LIN {X 0,Y 354.479,Z 638.418,A -85,B 0,C 180,E1 -13745.915,E2 -13745.915} C_VEL
LIN {X 0,Y 358.461,Z 680.686,A -85,B 0,C 180,E1 -13747.67,E2 -13747.67} C_VEL
LIN {X 0,Y 356.651,Z 726.677,A -85,B 0,C 180,E1 -13748.951,E2 -13748.951} C_VEL
LIN {X 0,Y 355.646,Z 740.597,A -85,B 0,C 180,E1 -13749.542,E2 -13749.542} C_VEL
LIN {X 0,Y 354.363,Z 753.48,A -85,B 0,C 180,E1 -13750.297,E2 -13750.297} C_VEL
LIN {X 0,Y 352.622,Z 767.795,A -85,B 0,C 180,E1 -13751.405,E2 -13751.405} C_VEL
LIN {X 0,Y 351.171,Z 779.191,A -85,B 0,C 180,E1 -13752.531,E2 -13752.531} C_VEL
LIN {X 0,Y 349.769,Z 790.795,A -85,B 0,C 180,E1 -13753.962,E2 -13753.962} C_VEL
LIN {X 0,Y 348.561,Z 801.445,A -85,B 0,C 180,E1 -13755.583,E2 -13755.583} C_VEL
LIN {X 0,Y 347.802,Z 809.876,A -85,B 0,C 180,E1 -13757.158,E2 -13757.158} C_VEL
LIN {X 0,Y 347.231,Z 817.648,A -85,B 0,C 180,E1 -13758.915,E2 -13758.915} C_VEL
LIN {X 0,Y 347.018,Z 823.966,A -85,B 0,C 180,E1 -13760.677,E2 -13760.677} C_VEL
LIN {X 0,Y 347.018,Z 831.536,A -85,B 0,C 180,E1 -13763.321,E2 -13763.321} C_VEL
LIN {X 0,Y 347.321,Z 835.911,A -85,B 0,C 180,E1 -13765.358,E2 -13765.358} C_VEL
LIN {X 0,Y 347.318,Z 837.708,A -85,B 0,C 180,E1 -13766.52,E2 -13766.52} C_VEL
LIN {X 0,Y 347.353,Z 838.988,A -85,B 0,C 180,E1 -13767.682,E2 -13767.682} C_VEL
LIN {X 0,Y 347.487,Z 839.813,A -85,B 0,C 180,E1 -13768.842,E2 -13768.842} C_VEL
LIN {X 0,Y 347.688,Z 840.196,A -85,B 0,C 180,E1 -13770.001,E2 -13770.001} C_VEL
LIN {X 0,Y 347.364,Z 840.046,A -85,B 0,C 180,E1 -13771.16,E2 -13771.16} C_VEL
LIN {X 0,Y 347.277,Z 839.445,A -85,B 0,C 180,E1 -13772.32,E2 -13772.32} C_VEL
LIN {X 0,Y 347.224,Z 838.385,A -85,B 0,C 180,E1 -13773.482,E2 -13773.482} C_VEL
LIN {X 0,Y 347.158,Z 836.872,A -85,B 0,C 180,E1 -13774.645,E2 -13774.645} C_VEL
LIN {X 0,Y 346.924,Z 833.32,A -85,B 0,C 180,E1 -13776.582,E2 -13776.582} C_VEL
LIN {X 0,Y 346.84,Z 827.807,A -85,B 0,C 180,E1 -13778.742,E2 -13778.742} C_VEL
LIN {X 0,Y 347.027,Z 820.861,A -85,B 0,C 180,E1 -13780.798,E2 -13780.798} C_VEL
LIN {X 0,Y 347.607,Z 813.484,A -85,B 0,C 180,E1 -13782.554,E2 -13782.554} C_VEL
LIN {X 0,Y 348.199,Z 805.239,A -85,B 0,C 180,E1 -13784.184,E2 -13784.184} C_VEL
LIN {X 0,Y 349.492,Z 795.668,A -85,B 0,C 180,E1 -13785.753,E2 -13785.753} C_VEL
LIN {X 0,Y 350.936,Z 785.164,A -85,B 0,C 180,E1 -13787.182,E2 -13787.182} C_VEL
LIN {X 0,Y 352.74,Z 772.484,A -85,B 0,C 180,E1 -13788.59,E2 -13788.59} C_VEL
LIN {X 0,Y 354.368,Z 760.134,A -85,B 0,C 180,E1 -13789.704,E2 -13789.704} C_VEL
LIN {X 0,Y 356.324,Z 745.84,A -85,B 0,C 180,E1 -13790.72,E2 -13790.72} C_VEL
LIN {X 0,Y 358.072,Z 729.548,A -85,B 0,C 180,E1 -13791.594,E2 -13791.594} C_VEL
LIN {X 0,Y 359.248,Z 714.539,A -85,B 0,C 180,E1 -13792.171,E2 -13792.171} C_VEL
LIN {X 0,Y 360.847,Z 679.966,A -85,B 0,C 180,E1 -13793.198,E2 -13793.198} C_VEL
LIN {X 0,Y 359.795,Z 647.693,A -85,B 0,C 180,E1 -13794.475,E2 -13794.475} C_VEL
LIN {X 0,Y 358.265,Z 629.878,A -85,B 0,C 180,E1 -13795.336,E2 -13795.336} C_VEL
LIN {X 0,Y 355.685,Z 611.993,A -85,B 0,C 180,E1 -13796.387,E2 -13796.387} C_VEL
LIN {X 0,Y 353.303,Z 598.764,A -85,B 0,C 180,E1 -13797.284,E2 -13797.284} C_VEL
LIN {X 0,Y 350.384,Z 585.333,A -85,B 0,C 180,E1 -13798.328,E2 -13798.328} C_VEL
LIN {X 0,Y 349.237,Z 579.78,A -85,B 0,C 180,E1 -13798.781,E2 -13798.781} C_VEL
LIN {X 0,Y 349.199,Z 578.981,A -85,B 0,C 180,E1 -13798.884,E2 -13798.884} C_VEL
LIN {X 0,Y 349.844,Z 568.142,A -85,B 0,C 180,E1 -13801.488,E2 -13801.488} C_VEL
LIN {X 0,Y 347.976,Z 557.739,A -85,B 0,C 180,E1 -13804.286,E2 -13804.286} C_VEL
LIN {X 0,Y 347.852,Z 557.158,A -85,B 0,C 180,E1 -13804.452,E2 -13804.452} C_VEL
LIN {X 0,Y 347.778,Z 557.162,A -85,B 0,C 180,E1 -13807.989,E2 -13807.989} C_VEL
LIN {X 0,Y 347.755,Z 557.164,A -85,B 0,C 180,E1 -13811.83,E2 -13811.83} C_VEL
LIN {X 0,Y 347.71,Z 557.174,A -85,B 0,C 180,E1 -13815.027,E2 -13815.027} C_VEL
LIN {X 0,Y 347.755,Z 557.165,A -85,B 0,C 180,E1 -13818.397,E2 -13818.397} C_VEL
LIN {X 0,Y 347.778,Z 557.163,A -85,B 0,C 180,E1 -13822.011,E2 -13822.011} C_VEL
LIN {X 0,Y 347.749,Z 557.169,A -85,B 0,C 180,E1 -13825.536,E2 -13825.536} C_VEL
LIN {X 0,Y 347.749,Z 557.167,A -85,B 0,C 180,E1 -13828.3,E2 -13828.3} C_VEL
LIN {X 0,Y 347.825,Z 557.277,A -85,B 0,C 180,E1 -13831.453,E2 -13831.453} C_VEL
LIN {X 0,Y 348.808,Z 559.969,A -85,B 0,C 180,E1 -13831.741,E2 -13831.741} C_VEL
LIN {X 0,Y 351.052,Z 562.747,A -85,B 0,C 180,E1 -13832.234,E2 -13832.234} C_VEL
LIN {X 0,Y 353.196,Z 565.986,A -85,B 0,C 180,E1 -13832.701,E2 -13832.701} C_VEL
LIN {X 0,Y 358.206,Z 574.137,A -85,B 0,C 180,E1 -13833.732,E2 -13833.732} C_VEL
LIN {X 0,Y 363.446,Z 583.854,A -85,B 0,C 180,E1 -13834.746,E2 -13834.746} C_VEL
LIN {X 0,Y 365.343,Z 588.205,A -85,B 0,C 180,E1 -13835.107,E2 -13835.107} C_VEL
LIN {X 0,Y 364.896,Z 614.714,A -85,B 0,C 180,E1 -13835.837,E2 -13835.837} C_VEL
LIN {X 0,Y 364.662,Z 629.49,A -85,B 0,C 180,E1 -13836.415,E2 -13836.415} C_VEL
LIN {X 0,Y 364.052,Z 644.188,A -85,B 0,C 180,E1 -13837.22,E2 -13837.22} C_VEL
LIN {X 0,Y 363.117,Z 657.203,A -85,B 0,C 180,E1 -13838.155,E2 -13838.155} C_VEL
LIN {X 0,Y 361.975,Z 669.32,A -85,B 0,C 180,E1 -13839.249,E2 -13839.249} C_VEL
LIN {X 0,Y 360.436,Z 681.905,A -85,B 0,C 180,E1 -13840.641,E2 -13840.641} C_VEL
LIN {X 0,Y 358.957,Z 692.336,A -85,B 0,C 180,E1 -13842.039,E2 -13842.039} C_VEL
LIN {X 0,Y 357.274,Z 702.674,A -85,B 0,C 180,E1 -13843.721,E2 -13843.721} C_VEL
LIN {X 0,Y 355.557,Z 712.086,A -85,B 0,C 180,E1 -13845.593,E2 -13845.593} C_VEL
LIN {X 0,Y 353.869,Z 720.615,A -85,B 0,C 180,E1 -13847.672,E2 -13847.672} C_VEL
LIN {X 0,Y 352.478,Z 727.173,A -85,B 0,C 180,E1 -13849.662,E2 -13849.662} C_VEL
LIN {X 0,Y 351.014,Z 733.098,A -85,B 0,C 180,E1 -13851.943,E2 -13851.943} C_VEL
LIN {X 0,Y 350.103,Z 737.454,A -85,B 0,C 180,E1 -13854.239,E2 -13854.239} C_VEL
LIN {X 0,Y 349.236,Z 740.513,A -85,B 0,C 180,E1 -13856.538,E2 -13856.538} C_VEL
LIN {X 0,Y 348.701,Z 742.261,A -85,B 0,C 180,E1 -13858.845,E2 -13858.845} C_VEL
LIN {X 0,Y 348.344,Z 742.765,A -85,B 0,C 180,E1 -13861.156,E2 -13861.156} C_VEL
LIN {X 0,Y 348.06,Z 742.044,A -85,B 0,C 180,E1 -13863.472,E2 -13863.472} C_VEL
LIN {X 0,Y 348.044,Z 740.07,A -85,B 0,C 180,E1 -13865.794,E2 -13865.794} C_VEL
LIN {X 0,Y 348.199,Z 738.597,A -85,B 0,C 180,E1 -13866.955,E2 -13866.955} C_VEL
LIN {X 0,Y 348.351,Z 734.679,A -85,B 0,C 180,E1 -13869.288,E2 -13869.288} C_VEL
LIN {X 0,Y 348.678,Z 729.336,A -85,B 0,C 180,E1 -13871.628,E2 -13871.628} C_VEL
LIN {X 0,Y 349.239,Z 722.409,A -85,B 0,C 180,E1 -13873.974,E2 -13873.974} C_VEL
LIN {X 0,Y 349.954,Z 714.96,A -85,B 0,C 180,E1 -13875.999,E2 -13875.999} C_VEL
LIN {X 0,Y 350.859,Z 705.636,A -85,B 0,C 180,E1 -13878.087,E2 -13878.087} C_VEL
LIN {X 0,Y 351.878,Z 695.29,A -85,B 0,C 180,E1 -13880,E2 -13880} C_VEL
LIN {X 0,Y 352.954,Z 683.746,A -85,B 0,C 180,E1 -13881.768,E2 -13881.768} C_VEL
LIN {X 0,Y 354.106,Z 670.886,A -85,B 0,C 180,E1 -13883.387,E2 -13883.387} C_VEL
LIN {X 0,Y 355.051,Z 658.101,A -85,B 0,C 180,E1 -13884.718,E2 -13884.718} C_VEL
LIN {X 0,Y 356.033,Z 644.114,A -85,B 0,C 180,E1 -13885.896,E2 -13885.896} C_VEL
LIN {X 0,Y 356.796,Z 629.668,A -85,B 0,C 180,E1 -13886.859,E2 -13886.859} C_VEL
LIN {X 0,Y 357.368,Z 614.609,A -85,B 0,C 180,E1 -13887.621,E2 -13887.621} C_VEL
LIN {X 0,Y 357.586,Z 599.377,A -85,B 0,C 180,E1 -13888.166,E2 -13888.166} C_VEL
LIN {X 0,Y 357.616,Z 583.757,A -85,B 0,C 180,E1 -13888.584,E2 -13888.584} C_VEL
LIN {X 0,Y 347.819,Z 557.232,A -85,B 0,C 180,E1 -13889.822,E2 -13889.822} C_VEL
LIN {X 0,Y 347.749,Z 557.17,A -85,B 0,C 180,E1 -13894.043,E2 -13894.043} C_VEL
LIN {X 0,Y 347.762,Z 557.162,A -85,B 0,C 180,E1 -13897.32,E2 -13897.32} C_VEL
LIN {X 0,Y 347.733,Z 557.172,A -85,B 0,C 180,E1 -13900.296,E2 -13900.296} C_VEL
LIN {X 0,Y 347.723,Z 557.167,A -85,B 0,C 180,E1 -13903.407,E2 -13903.407} C_VEL
LIN {X 0,Y 347.725,Z 557.17,A -85,B 0,C 180,E1 -13906.685,E2 -13906.685} C_VEL
LIN {X 0,Y 347.747,Z 557.168,A -85,B 0,C 180,E1 -13910.172,E2 -13910.172} C_VEL
LIN {X 0,Y 347.766,Z 557.166,A -85,B 0,C 180,E1 -13912.679,E2 -13912.679} C_VEL
LIN {X 0,Y 347.748,Z 557.165,A -85,B 0,C 180,E1 -13915.955,E2 -13915.955} C_VEL
LIN {X 0,Y 347.748,Z 557.164,A -85,B 0,C 180,E1 -13919.651,E2 -13919.651} C_VEL
LIN {X 0,Y 347.83,Z 557.154,A -85,B 0,C 180,E1 -13923.607,E2 -13923.607} C_VEL
LIN {X 0,Y 347.788,Z 557.161,A -85,B 0,C 180,E1 -13926.161,E2 -13926.161} C_VEL
LIN {X 0,Y 347.811,Z 557.156,A -85,B 0,C 180,E1 -13929.909,E2 -13929.909} C_VEL
LIN {X 0,Y 347.865,Z 557.152,A -85,B 0,C 180,E1 -13932.359,E2 -13932.359} C_VEL
LIN {X 0,Y 347.896,Z 557.146,A -85,B 0,C 180,E1 -13935.97,E2 -13935.97} C_VEL
LIN {X 0,Y 347.927,Z 557.143,A -85,B 0,C 180,E1 -13939.525,E2 -13939.525} C_VEL
LIN {X 0,Y 348.072,Z 557.124,A -85,B 0,C 180,E1 -13941.874,E2 -13941.874} C_VEL
LIN {X 0,Y 348.066,Z 557.125,A -85,B 0,C 180,E1 -13944.205,E2 -13944.205} C_VEL
LIN {X 0,Y 348.206,Z 557.108,A -85,B 0,C 180,E1 -13947.686,E2 -13947.686} C_VEL
LIN {X 0,Y 348.344,Z 557.09,A -85,B 0,C 180,E1 -13949.999,E2 -13949.999} C_VEL
LIN {X 0,Y 348.206,Z 557.107,A -85,B 0,C 180,E1 -13952.313,E2 -13952.313} C_VEL
LIN {X 0,Y 348.101,Z 557.123,A -85,B 0,C 180,E1 -13956.957,E2 -13956.957} C_VEL
LIN {X 0,Y 347.965,Z 557.144,A -85,B 0,C 180,E1 -13959.298,E2 -13959.298} C_VEL
LIN {X 0,Y 347.891,Z 557.148,A -85,B 0,C 180,E1 -13962.839,E2 -13962.839} C_VEL
LIN {X 0,Y 347.836,Z 557.153,A -85,B 0,C 180,E1 -13966.431,E2 -13966.431} C_VEL
LIN {X 0,Y 347.847,Z 557.153,A -85,B 0,C 180,E1 -13968.86,E2 -13968.86} C_VEL
LIN {X 0,Y 347.771,Z 557.161,A -85,B 0,C 180,E1 -13972.579,E2 -13972.579} C_VEL
LIN {X 0,Y 347.808,Z 557.158,A -85,B 0,C 180,E1 -13975.108,E2 -13975.108} C_VEL
LIN {X 0,Y 347.808,Z 557.163,A -85,B 0,C 180,E1 -13977.693,E2 -13977.693} C_VEL
LIN {X 0,Y 347.767,Z 557.163,A -85,B 0,C 180,E1 -13980.345,E2 -13980.345} C_VEL
LIN {X 0,Y 347.743,Z 557.168,A -85,B 0,C 180,E1 -13984.043,E2 -13984.043} C_VEL
LIN {X 0,Y 347.761,Z 557.164,A -85,B 0,C 180,E1 -13987.32,E2 -13987.32} C_VEL
LIN {X 0,Y 347.75,Z 557.166,A -85,B 0,C 180,E1 -13990.294,E2 -13990.294} C_VEL
LIN {X 0,Y 347.764,Z 557.164,A -85,B 0,C 180,E1 -13993.401,E2 -13993.401} C_VEL
LIN {X 0,Y 347.809,Z 557.157,A -85,B 0,C 180,E1 -13996.67,E2 -13996.67} C_VEL
LIN {X 0,Y 347.78,Z 557.165,A -85,B 0,C 180,E1 -14000.123,E2 -14000.123} C_VEL
LIN {X 0,Y 347.68,Z 557.818,A -85,B 0,C 180,E1 -14000.73,E2 -14000.73} C_VEL
LIN {X 0,Y 347.391,Z 559.998,A -85,B 0,C 180,E1 -14001.422,E2 -14001.422} C_VEL
LIN {X 0,Y 347.087,Z 563.175,A -85,B 0,C 180,E1 -14002.021,E2 -14002.021} C_VEL
LIN {X 0,Y 346.917,Z 567.944,A -85,B 0,C 180,E1 -14002.622,E2 -14002.622} C_VEL
LIN {X 0,Y 347.234,Z 573.312,A -85,B 0,C 180,E1 -14003.094,E2 -14003.094} C_VEL
LIN {X 0,Y 348.465,Z 578.915,A -85,B 0,C 180,E1 -14003.416,E2 -14003.416} C_VEL
LIN {X 0,Y 349.772,Z 582.501,A -85,B 0,C 180,E1 -14003.573,E2 -14003.573} C_VEL
LIN {X 0,Y 349.053,Z 620.126,A -85,B 0,C 180,E1 -14004.541,E2 -14004.541} C_VEL
LIN {X 0,Y 348.82,Z 634.327,A -85,B 0,C 180,E1 -14005.132,E2 -14005.132} C_VEL
LIN {X 0,Y 348.195,Z 648.532,A -85,B 0,C 180,E1 -14005.963,E2 -14005.963} C_VEL
LIN {X 0,Y 347.478,Z 660.802,A -85,B 0,C 180,E1 -14006.901,E2 -14006.901} C_VEL
LIN {X 0,Y 346.554,Z 674.042,A -85,B 0,C 180,E1 -14008.179,E2 -14008.179} C_VEL
LIN {X 0,Y 345.474,Z 685.971,A -85,B 0,C 180,E1 -14009.601,E2 -14009.601} C_VEL
LIN {X 0,Y 344.643,Z 696.152,A -85,B 0,C 180,E1 -14011.089,E2 -14011.089} C_VEL
LIN {X 0,Y 343.596,Z 706.515,A -85,B 0,C 180,E1 -14012.929,E2 -14012.929} C_VEL
LIN {X 0,Y 342.781,Z 715.232,A -85,B 0,C 180,E1 -14014.822,E2 -14014.822} C_VEL
LIN {X 0,Y 342.118,Z 722.337,A -85,B 0,C 180,E1 -14016.707,E2 -14016.707} C_VEL
LIN {X 0,Y 341.513,Z 728.954,A -85,B 0,C 180,E1 -14018.892,E2 -14018.892} C_VEL
LIN {X 0,Y 341.151,Z 733.355,A -85,B 0,C 180,E1 -14020.755,E2 -14020.755} C_VEL
LIN {X 0,Y 340.967,Z 735.707,A -85,B 0,C 180,E1 -14021.991,E2 -14021.991} C_VEL
LIN {X 0,Y 340.772,Z 739.15,A -85,B 0,C 180,E1 -14024.449,E2 -14024.449} C_VEL
LIN {X 0,Y 340.83,Z 741.068,A -85,B 0,C 180,E1 -14026.89,E2 -14026.89} C_VEL
LIN {X 0,Y 340.94,Z 741.459,A -85,B 0,C 180,E1 -14028.105,E2 -14028.105} C_VEL
LIN {X 0,Y 341.317,Z 741.079,A -85,B 0,C 180,E1 -14030.519,E2 -14030.519} C_VEL
LIN {X 0,Y 341.831,Z 739.281,A -85,B 0,C 180,E1 -14032.915,E2 -14032.915} C_VEL
LIN {X 0,Y 342.719,Z 735.987,A -85,B 0,C 180,E1 -14035.295,E2 -14035.295} C_VEL
LIN {X 0,Y 343.442,Z 732.461,A -85,B 0,C 180,E1 -14037.068,E2 -14037.068} C_VEL
LIN {X 0,Y 344.428,Z 727.73,A -85,B 0,C 180,E1 -14038.915,E2 -14038.915} C_VEL
LIN {X 0,Y 345.636,Z 721.395,A -85,B 0,C 180,E1 -14040.874,E2 -14040.874} C_VEL
LIN {X 0,Y 346.918,Z 714.409,A -85,B 0,C 180,E1 -14042.613,E2 -14042.613} C_VEL
LIN {X 0,Y 348.453,Z 705.922,A -85,B 0,C 180,E1 -14044.338,E2 -14044.338} C_VEL
LIN {X 0,Y 349.884,Z 695.604,A -85,B 0,C 180,E1 -14046.054,E2 -14046.054} C_VEL
LIN {X 0,Y 351.355,Z 684.983,A -85,B 0,C 180,E1 -14047.471,E2 -14047.471} C_VEL
LIN {X 0,Y 352.66,Z 673.304,A -85,B 0,C 180,E1 -14048.741,E2 -14048.741} C_VEL
LIN {X 0,Y 353.818,Z 660.233,A -85,B 0,C 180,E1 -14049.865,E2 -14049.865} C_VEL
LIN {X 0,Y 354.55,Z 647.65,A -85,B 0,C 180,E1 -14050.71,E2 -14050.71} C_VEL
LIN {X 0,Y 355.091,Z 633.242,A -85,B 0,C 180,E1 -14051.416,E2 -14051.416} C_VEL
LIN {X 0,Y 355.244,Z 618.147,A -85,B 0,C 180,E1 -14051.899,E2 -14051.899} C_VEL
LIN {X 0,Y 356.085,Z 586.597,A -85,B 0,C 180,E1 -14052.724,E2 -14052.724} C_VEL
LIN {X 0,Y 350.383,Z 575.035,A -85,B 0,C 180,E1 -14053.751,E2 -14053.751} C_VEL
LIN {X 0,Y 345.203,Z 565.966,A -85,B 0,C 180,E1 -14054.718,E2 -14054.718} C_VEL
LIN {X 0,Y 342.724,Z 562.055,A -85,B 0,C 180,E1 -14055.194,E2 -14055.194} C_VEL
LIN {X 0,Y 341.147,Z 559.521,A -85,B 0,C 180,E1 -14055.509,E2 -14055.509} C_VEL
LIN {X 0,Y 340.8,Z 558.041,A -85,B 0,C 180,E1 -14055.628,E2 -14055.628} C_VEL
LIN {X 0,Y 340.835,Z 558.032,A -85,B 0,C 180,E1 -14058.468,E2 -14058.468} C_VEL
LIN {X 0,Y 340.751,Z 558.039,A -85,B 0,C 180,E1 -14061.858,E2 -14061.858} C_VEL
LIN {X 0,Y 340.77,Z 558.033,A -85,B 0,C 180,E1 -14065.665,E2 -14065.665} C_VEL
LIN {X 0,Y 340.74,Z 558.035,A -85,B 0,C 180,E1 -14068.32,E2 -14068.32} C_VEL
LIN {X 0,Y 340.702,Z 558.04,A -85,B 0,C 180,E1 -14071.045,E2 -14071.045} C_VEL
LIN {X 0,Y 340.716,Z 558.036,A -85,B 0,C 180,E1 -14075.28,E2 -14075.28} C_VEL
LIN {X 0,Y 340.708,Z 558.041,A -85,B 0,C 180,E1 -14078.387,E2 -14078.387} C_VEL
LIN {X 0,Y 340.698,Z 558.041,A -85,B 0,C 180,E1 -14082.046,E2 -14082.046} C_VEL
LIN {X 0,Y 340.683,Z 558.049,A -85,B 0,C 180,E1 -14085.462,E2 -14085.462} C_VEL
LIN {X 0,Y 340.685,Z 558.038,A -85,B 0,C 180,E1 -14088.691,E2 -14088.691} C_VEL
LIN {X 0,Y 340.791,Z 558.206,A -85,B 0,C 180,E1 -14090.841,E2 -14090.841} C_VEL
LIN {X 0,Y 343.738,Z 572.66,A -85,B 0,C 180,E1 -14094.869,E2 -14094.869} C_VEL
LIN {X 0,Y 345.677,Z 582.119,A -85,B 0,C 180,E1 -14097.401,E2 -14097.401} C_VEL
LIN {X 0,Y 343.823,Z 598.712,A -85,B 0,C 180,E1 -14101.517,E2 -14101.517} C_VEL
LIN {X 0,Y 343.038,Z 606.504,A -85,B 0,C 180,E1 -14103.432,E2 -14103.432} C_VEL
LIN {X 0,Y 343.793,Z 611.517,A -85,B 0,C 180,E1 -14103.734,E2 -14103.734} C_VEL
LIN {X 0,Y 346.795,Z 628.501,A -85,B 0,C 180,E1 -14104.725,E2 -14104.725} C_VEL
LIN {X 0,Y 348.814,Z 642.749,A -85,B 0,C 180,E1 -14105.451,E2 -14105.451} C_VEL
LIN {X 0,Y 352.306,Z 681.851,A -85,B 0,C 180,E1 -14107.128,E2 -14107.128} C_VEL
LIN {X 0,Y 350.412,Z 725.147,A -85,B 0,C 180,E1 -14108.375,E2 -14108.375} C_VEL
LIN {X 0,Y 349.29,Z 739.422,A -85,B 0,C 180,E1 -14108.999,E2 -14108.999} C_VEL
LIN {X 0,Y 347.923,Z 752.223,A -85,B 0,C 180,E1 -14109.763,E2 -14109.763} C_VEL
LIN {X 0,Y 346.145,Z 766.523,A -85,B 0,C 180,E1 -14110.89,E2 -14110.89} C_VEL
LIN {X 0,Y 344.396,Z 779.089,A -85,B 0,C 180,E1 -14112.176,E2 -14112.176} C_VEL
LIN {X 0,Y 342.911,Z 790.465,A -85,B 0,C 180,E1 -14113.633,E2 -14113.633} C_VEL
LIN {X 0,Y 341.667,Z 800.921,A -85,B 0,C 180,E1 -14115.286,E2 -14115.286} C_VEL
LIN {X 0,Y 340.713,Z 810.655,A -85,B 0,C 180,E1 -14117.189,E2 -14117.189} C_VEL
LIN {X 0,Y 340.11,Z 818.061,A -85,B 0,C 180,E1 -14118.981,E2 -14118.981} C_VEL
LIN {X 0,Y 339.919,Z 824.947,A -85,B 0,C 180,E1 -14121.08,E2 -14121.08} C_VEL
LIN {X 0,Y 339.954,Z 829.615,A -85,B 0,C 180,E1 -14122.9,E2 -14122.9} C_VEL
LIN {X 0,Y 340.286,Z 834.615,A -85,B 0,C 180,E1 -14125.262,E2 -14125.262} C_VEL
LIN {X 0,Y 340.299,Z 836.454,A -85,B 0,C 180,E1 -14126.449,E2 -14126.449} C_VEL
LIN {X 0,Y 340.333,Z 837.808,A -85,B 0,C 180,E1 -14127.634,E2 -14127.634} C_VEL
LIN {X 0,Y 340.475,Z 838.671,A -85,B 0,C 180,E1 -14128.818,E2 -14128.818} C_VEL
LIN {X 0,Y 340.677,Z 839.086,A -85,B 0,C 180,E1 -14130.001,E2 -14130.001} C_VEL
LIN {X 0,Y 340.364,Z 838.97,A -85,B 0,C 180,E1 -14131.184,E2 -14131.184} C_VEL
LIN {X 0,Y 340.235,Z 838.427,A -85,B 0,C 180,E1 -14132.368,E2 -14132.368} C_VEL
LIN {X 0,Y 340.177,Z 837.403,A -85,B 0,C 180,E1 -14133.554,E2 -14133.554} C_VEL
LIN {X 0,Y 340.09,Z 835.918,A -85,B 0,C 180,E1 -14134.742,E2 -14134.742} C_VEL
LIN {X 0,Y 339.823,Z 832.009,A -85,B 0,C 180,E1 -14136.921,E2 -14136.921} C_VEL
LIN {X 0,Y 339.758,Z 827.001,A -85,B 0,C 180,E1 -14138.926,E2 -14138.926} C_VEL
LIN {X 0,Y 340.005,Z 820.192,A -85,B 0,C 180,E1 -14141.023,E2 -14141.023} C_VEL
LIN {X 0,Y 340.605,Z 812.925,A -85,B 0,C 180,E1 -14142.816,E2 -14142.816} C_VEL
LIN {X 0,Y 341.448,Z 803.786,A -85,B 0,C 180,E1 -14144.669,E2 -14144.669} C_VEL
LIN {X 0,Y 342.844,Z 793.537,A -85,B 0,C 180,E1 -14146.372,E2 -14146.372} C_VEL
LIN {X 0,Y 344.724,Z 781.722,A -85,B 0,C 180,E1 -14147.961,E2 -14147.961} C_VEL
LIN {X 0,Y 346.663,Z 768.673,A -85,B 0,C 180,E1 -14149.389,E2 -14149.389} C_VEL
LIN {X 0,Y 348.566,Z 755.933,A -85,B 0,C 180,E1 -14150.508,E2 -14150.508} C_VEL
LIN {X 0,Y 350.597,Z 740.936,A -85,B 0,C 180,E1 -14151.537,E2 -14151.537} C_VEL
LIN {X 0,Y 352.261,Z 725.307,A -85,B 0,C 180,E1 -14152.354,E2 -14152.354} C_VEL
LIN {X 0,Y 353.561,Z 708.761,A -85,B 0,C 180,E1 -14152.961,E2 -14152.961} C_VEL
LIN {X 0,Y 354.931,Z 680.758,A -85,B 0,C 180,E1 -14153.817,E2 -14153.817} C_VEL
LIN {X 0,Y 354.104,Z 649.055,A -85,B 0,C 180,E1 -14155.113,E2 -14155.113} C_VEL
LIN {X 0,Y 352.529,Z 629.953,A -85,B 0,C 180,E1 -14156.084,E2 -14156.084} C_VEL
LIN {X 0,Y 350.062,Z 612.121,A -85,B 0,C 180,E1 -14157.188,E2 -14157.188} C_VEL
LIN {X 0,Y 346.975,Z 595.359,A -85,B 0,C 180,E1 -14158.429,E2 -14158.429} C_VEL
LIN {X 0,Y 345.443,Z 588.209,A -85,B 0,C 180,E1 -14159.037,E2 -14159.037} C_VEL
LIN {X 0,Y 343.995,Z 581.651,A -85,B 0,C 180,E1 -14159.618,E2 -14159.618} C_VEL
LIN {X 0,Y 342.667,Z 575.729,A -85,B 0,C 180,E1 -14160.166,E2 -14160.166} C_VEL
LIN {X 0,Y 342.615,Z 574.666,A -85,B 0,C 180,E1 -14160.286,E2 -14160.286} C_VEL
LIN {X 0,Y 342.808,Z 568.394,A -85,B 0,C 180,E1 -14161.865,E2 -14161.865} C_VEL
LIN {X 0,Y 340.804,Z 558.035,A -85,B 0,C 180,E1 -14164.76,E2 -14164.76} C_VEL
LIN {X 0,Y 340.714,Z 558.042,A -85,B 0,C 180,E1 -14168.386,E2 -14168.386} C_VEL
LIN {X 0,Y 340.703,Z 558.042,A -85,B 0,C 180,E1 -14172.046,E2 -14172.046} C_VEL
LIN {X 0,Y 340.656,Z 558.049,A -85,B 0,C 180,E1 -14176.227,E2 -14176.227} C_VEL
LIN {X 0,Y 340.693,Z 558.047,A -85,B 0,C 180,E1 -14179.753,E2 -14179.753} C_VEL
LIN {X 0,Y 340.71,Z 558.046,A -85,B 0,C 180,E1 -14183.258,E2 -14183.258} C_VEL
LIN {X 0,Y 340.697,Z 558.045,A -85,B 0,C 180,E1 -14186.153,E2 -14186.153} C_VEL
LIN {X 0,Y 340.749,Z 558.104,A -85,B 0,C 180,E1 -14190.108,E2 -14190.108} C_VEL
LIN {X 0,Y 341.571,Z 560.593,A -85,B 0,C 180,E1 -14190.396,E2 -14190.396} C_VEL
LIN {X 0,Y 343.716,Z 562.98,A -85,B 0,C 180,E1 -14190.929,E2 -14190.929} C_VEL
LIN {X 0,Y 346.293,Z 566.945,A -85,B 0,C 180,E1 -14191.573,E2 -14191.573} C_VEL
LIN {X 0,Y 347.729,Z 569.144,A -85,B 0,C 180,E1 -14191.924,E2 -14191.924} C_VEL
LIN {X 0,Y 351.755,Z 575.273,A -85,B 0,C 180,E1 -14192.808,E2 -14192.808} C_VEL
LIN {X 0,Y 357.606,Z 585.832,A -85,B 0,C 180,E1 -14194.027,E2 -14194.027} C_VEL
LIN {X 0,Y 359.713,Z 590.39,A -85,B 0,C 180,E1 -14194.465,E2 -14194.465} C_VEL
LIN {X 0,Y 359.245,Z 616.254,A -85,B 0,C 180,E1 -14195.201,E2 -14195.201} C_VEL
LIN {X 0,Y 358.99,Z 630.424,A -85,B 0,C 180,E1 -14195.763,E2 -14195.763} C_VEL
LIN {X 0,Y 358.33,Z 644.211,A -85,B 0,C 180,E1 -14196.522,E2 -14196.522} C_VEL
LIN {X 0,Y 357.228,Z 658.781,A -85,B 0,C 180,E1 -14197.578,E2 -14197.578} C_VEL
LIN {X 0,Y 355.873,Z 671.946,A -85,B 0,C 180,E1 -14198.791,E2 -14198.791} C_VEL
LIN {X 0,Y 354.332,Z 683.78,A -85,B 0,C 180,E1 -14200.143,E2 -14200.143} C_VEL
LIN {X 0,Y 352.874,Z 693.116,A -85,B 0,C 180,E1 -14201.417,E2 -14201.417} C_VEL
LIN {X 0,Y 351.129,Z 703.543,A -85,B 0,C 180,E1 -14203.128,E2 -14203.128} C_VEL
LIN {X 0,Y 349.401,Z 712.523,A -85,B 0,C 180,E1 -14204.906,E2 -14204.906} C_VEL
LIN {X 0,Y 347.675,Z 720.581,A -85,B 0,C 180,E1 -14206.855,E2 -14206.855} C_VEL
LIN {X 0,Y 346.13,Z 727.356,A -85,B 0,C 180,E1 -14208.878,E2 -14208.878} C_VEL
LIN {X 0,Y 344.551,Z 733.524,A -85,B 0,C 180,E1 -14211.2,E2 -14211.2} C_VEL
LIN {X 0,Y 343.786,Z 737.075,A -85,B 0,C 180,E1 -14212.954,E2 -14212.954} C_VEL
LIN {X 0,Y 342.781,Z 740.635,A -85,B 0,C 180,E1 -14215.295,E2 -14215.295} C_VEL
LIN {X 0,Y 342.007,Z 742.879,A -85,B 0,C 180,E1 -14217.644,E2 -14217.644} C_VEL
LIN {X 0,Y 341.52,Z 743.875,A -85,B 0,C 180,E1 -14219.999,E2 -14219.999} C_VEL
LIN {X 0,Y 341.125,Z 743.639,A -85,B 0,C 180,E1 -14222.361,E2 -14222.361} C_VEL
LIN {X 0,Y 340.879,Z 742.161,A -85,B 0,C 180,E1 -14224.73,E2 -14224.73} C_VEL
LIN {X 0,Y 341.167,Z 739.375,A -85,B 0,C 180,E1 -14227.099,E2 -14227.099} C_VEL
LIN {X 0,Y 341.334,Z 735.295,A -85,B 0,C 180,E1 -14229.48,E2 -14229.48} C_VEL
LIN {X 0,Y 341.705,Z 729.78,A -85,B 0,C 180,E1 -14231.868,E2 -14231.868} C_VEL
LIN {X 0,Y 342.305,Z 722.666,A -85,B 0,C 180,E1 -14234.263,E2 -14234.263} C_VEL
LIN {X 0,Y 343.064,Z 714.899,A -85,B 0,C 180,E1 -14236.36,E2 -14236.36} C_VEL
LIN {X 0,Y 343.975,Z 705.438,A -85,B 0,C 180,E1 -14238.462,E2 -14238.462} C_VEL
LIN {X 0,Y 344.974,Z 695.688,A -85,B 0,C 180,E1 -14240.263,E2 -14240.263} C_VEL
LIN {X 0,Y 346.081,Z 683.947,A -85,B 0,C 180,E1 -14242.066,E2 -14242.066} C_VEL
LIN {X 0,Y 347.152,Z 672.207,A -85,B 0,C 180,E1 -14243.567,E2 -14243.567} C_VEL
LIN {X 0,Y 348.139,Z 659.504,A -85,B 0,C 180,E1 -14244.919,E2 -14244.919} C_VEL
LIN {X 0,Y 349.134,Z 645.52,A -85,B 0,C 180,E1 -14246.125,E2 -14246.125} C_VEL
LIN {X 0,Y 349.947,Z 631.172,A -85,B 0,C 180,E1 -14247.105,E2 -14247.105} C_VEL
LIN {X 0,Y 350.573,Z 615.386,A -85,B 0,C 180,E1 -14247.92,E2 -14247.92} C_VEL
LIN {X 0,Y 350.792,Z 600.111,A -85,B 0,C 180,E1 -14248.473,E2 -14248.473} C_VEL
LIN {X 0,Y 350.777,Z 585.152,A -85,B 0,C 180,E1 -14248.887,E2 -14248.887} C_VEL
LIN {X 0,Y 340.738,Z 558.042,A -85,B 0,C 180,E1 -14250.195,E2 -14250.195} C_VEL
LIN {X 0,Y 340.724,Z 558.043,A -85,B 0,C 180,E1 -14254.404,E2 -14254.404} C_VEL
LIN {X 0,Y 340.71,Z 558.045,A -85,B 0,C 180,E1 -14258.385,E2 -14258.385} C_VEL
LIN {X 0,Y 340.699,Z 558.046,A -85,B 0,C 180,E1 -14262.045,E2 -14262.045} C_VEL
LIN {X 0,Y 340.652,Z 558.053,A -85,B 0,C 180,E1 -14266.226,E2 -14266.226} C_VEL
LIN {X 0,Y 340.688,Z 558.044,A -85,B 0,C 180,E1 -14269.752,E2 -14269.752} C_VEL
LIN {X 0,Y 340.707,Z 558.042,A -85,B 0,C 180,E1 -14273.258,E2 -14273.258} C_VEL
LIN {X 0,Y 340.692,Z 558.046,A -85,B 0,C 180,E1 -14276.153,E2 -14276.153} C_VEL
LIN {X 0,Y 340.74,Z 558.041,A -85,B 0,C 180,E1 -14280.329,E2 -14280.329} C_VEL
LIN {X 0,Y 340.802,Z 558.032,A -85,B 0,C 180,E1 -14283.019,E2 -14283.019} C_VEL
LIN {X 0,Y 340.755,Z 558.035,A -85,B 0,C 180,E1 -14285.638,E2 -14285.638} C_VEL
LIN {X 0,Y 340.751,Z 558.036,A -85,B 0,C 180,E1 -14289.474,E2 -14289.474} C_VEL
LIN {X 0,Y 340.856,Z 558.023,A -85,B 0,C 180,E1 -14291.983,E2 -14291.983} C_VEL
LIN {X 0,Y 340.868,Z 558.021,A -85,B 0,C 180,E1 -14295.704,E2 -14295.704} C_VEL
LIN {X 0,Y 340.869,Z 558.024,A -85,B 0,C 180,E1 -14299.305,E2 -14299.305} C_VEL
LIN {X 0,Y 341.074,Z 558.001,A -85,B 0,C 180,E1 -14302.897,E2 -14302.897} C_VEL
LIN {X 0,Y 341.168,Z 557.985,A -85,B 0,C 180,E1 -14307.638,E2 -14307.638} C_VEL
LIN {X 0,Y 341.294,Z 557.968,A -85,B 0,C 180,E1 -14309.999,E2 -14309.999} C_VEL
LIN {X 0,Y 341.168,Z 557.984,A -85,B 0,C 180,E1 -14312.361,E2 -14312.361} C_VEL
LIN {X 0,Y 341.071,Z 558,A -85,B 0,C 180,E1 -14317.101,E2 -14317.101} C_VEL
LIN {X 0,Y 340.871,Z 558.022,A -85,B 0,C 180,E1 -14320.693,E2 -14320.693} C_VEL
LIN {X 0,Y 340.859,Z 558.022,A -85,B 0,C 180,E1 -14324.324,E2 -14324.324} C_VEL
LIN {X 0,Y 340.833,Z 558.026,A -85,B 0,C 180,E1 -14328.466,E2 -14328.466} C_VEL
LIN {X 0,Y 340.749,Z 558.039,A -85,B 0,C 180,E1 -14331.856,E2 -14331.856} C_VEL
LIN {X 0,Y 340.768,Z 558.04,A -85,B 0,C 180,E1 -14335.664,E2 -14335.664} C_VEL
LIN {X 0,Y 340.738,Z 558.038,A -85,B 0,C 180,E1 -14338.319,E2 -14338.319} C_VEL
LIN {X 0,Y 340.713,Z 558.041,A -85,B 0,C 180,E1 -14341.042,E2 -14341.042} C_VEL
LIN {X 0,Y 340.714,Z 558.042,A -85,B 0,C 180,E1 -14345.278,E2 -14345.278} C_VEL
LIN {X 0,Y 340.714,Z 558.042,A -85,B 0,C 180,E1 -14348.388,E2 -14348.388} C_VEL
LIN {X 0,Y 340.728,Z 558.044,A -85,B 0,C 180,E1 -14352.052,E2 -14352.052} C_VEL
LIN {X 0,Y 340.768,Z 558.035,A -85,B 0,C 180,E1 -14355.476,E2 -14355.476} C_VEL
LIN {X 0,Y 340.721,Z 558.04,A -85,B 0,C 180,E1 -14358.696,E2 -14358.696} C_VEL
LIN {X 0,Y 340.745,Z 558.12,A -85,B 0,C 180,E1 -14362.452,E2 -14362.452} C_VEL
LIN {X 0,Y 348.465,Z 578.915,A -85,B 0,C 180,E1 -14363.416,E2 -14363.416} C_VEL
LIN {X 0,Y 348.748,Z 582.061,A -85,B 0,C 180,E1 -14363.511,E2 -14363.511} C_VEL
LIN {X 0,Y 347.526,Z 586.511,A -85,B 0,C 180,E1 -14363.564,E2 -14363.564} C_VEL
LIN {X 0,Y 343.394,Z 595.307,A -85,B 0,C 180,E1 -14363.585,E2 -14363.585} C_VEL
LIN {X 0,Y 342.597,Z 599.34,A -85,B 0,C 180,E1 -14363.654,E2 -14363.654} C_VEL
LIN {X 0,Y 342.258,Z 623.08,A -85,B 0,C 180,E1 -14364.32,E2 -14364.32} C_VEL
LIN {X 0,Y 341.915,Z 637.381,A -85,B 0,C 180,E1 -14364.961,E2 -14364.961} C_VEL
LIN {X 0,Y 341.253,Z 651.172,A -85,B 0,C 180,E1 -14365.818,E2 -14365.818} C_VEL
LIN {X 0,Y 340.435,Z 663.815,A -85,B 0,C 180,E1 -14366.834,E2 -14366.834} C_VEL
LIN {X 0,Y 339.472,Z 677.102,A -85,B 0,C 180,E1 -14368.182,E2 -14368.182} C_VEL
LIN {X 0,Y 338.422,Z 688.301,A -85,B 0,C 180,E1 -14369.59,E2 -14369.59} C_VEL
LIN {X 0,Y 337.383,Z 699.842,A -85,B 0,C 180,E1 -14371.373,E2 -14371.373} C_VEL
LIN {X 0,Y 336.366,Z 710.057,A -85,B 0,C 180,E1 -14373.307,E2 -14373.307} C_VEL
LIN {X 0,Y 335.568,Z 718.306,A -85,B 0,C 180,E1 -14375.237,E2 -14375.237} C_VEL
LIN {X 0,Y 334.837,Z 725.926,A -85,B 0,C 180,E1 -14377.445,E2 -14377.445} C_VEL
LIN {X 0,Y 334.302,Z 732.054,A -85,B 0,C 180,E1 -14379.704,E2 -14379.704} C_VEL
LIN {X 0,Y 333.896,Z 737.09,A -85,B 0,C 180,E1 -14382.23,E2 -14382.23} C_VEL
LIN {X 0,Y 333.759,Z 739.77,A -85,B 0,C 180,E1 -14384.113,E2 -14384.113} C_VEL
LIN {X 0,Y 333.805,Z 741.917,A -85,B 0,C 180,E1 -14386.609,E2 -14386.609} C_VEL
LIN {X 0,Y 334.051,Z 742.593,A -85,B 0,C 180,E1 -14389.086,E2 -14389.086} C_VEL
LIN {X 0,Y 334.394,Z 742.055,A -85,B 0,C 180,E1 -14391.037,E2 -14391.037} C_VEL
LIN {X 0,Y 334.812,Z 740.822,A -85,B 0,C 180,E1 -14392.765,E2 -14392.765} C_VEL
LIN {X 0,Y 335.723,Z 737.752,A -85,B 0,C 180,E1 -14395.197,E2 -14395.197} C_VEL
LIN {X 0,Y 336.79,Z 733.158,A -85,B 0,C 180,E1 -14397.609,E2 -14397.609} C_VEL
LIN {X 0,Y 337.818,Z 728.567,A -85,B 0,C 180,E1 -14399.4,E2 -14399.4} C_VEL
LIN {X 0,Y 339.196,Z 721.866,A -85,B 0,C 180,E1 -14401.485,E2 -14401.485} C_VEL
LIN {X 0,Y 340.629,Z 714.712,A -85,B 0,C 180,E1 -14403.253,E2 -14403.253} C_VEL
LIN {X 0,Y 342.185,Z 706.013,A -85,B 0,C 180,E1 -14405.008,E2 -14405.008} C_VEL
LIN {X 0,Y 343.475,Z 697.358,A -85,B 0,C 180,E1 -14406.462,E2 -14406.462} C_VEL
LIN {X 0,Y 345.032,Z 686.902,A -85,B 0,C 180,E1 -14407.903,E2 -14407.903} C_VEL
LIN {X 0,Y 346.414,Z 675.463,A -85,B 0,C 180,E1 -14409.194,E2 -14409.194} C_VEL
LIN {X 0,Y 347.684,Z 662.682,A -85,B 0,C 180,E1 -14410.335,E2 -14410.335} C_VEL
LIN {X 0,Y 348.494,Z 649.235,A -85,B 0,C 180,E1 -14411.267,E2 -14411.267} C_VEL
LIN {X 0,Y 349.081,Z 635.588,A -85,B 0,C 180,E1 -14411.952,E2 -14411.952} C_VEL
LIN {X 0,Y 349.266,Z 620.697,A -85,B 0,C 180,E1 -14412.464,E2 -14412.464} C_VEL
LIN {X 0,Y 350.208,Z 588.836,A -85,B 0,C 180,E1 -14413.333,E2 -14413.333} C_VEL
LIN {X 0,Y 344.803,Z 578.024,A -85,B 0,C 180,E1 -14414.354,E2 -14414.354} C_VEL
LIN {X 0,Y 338.545,Z 567.292,A -85,B 0,C 180,E1 -14415.598,E2 -14415.598} C_VEL
LIN {X 0,Y 335.901,Z 563.186,A -85,B 0,C 180,E1 -14416.153,E2 -14416.153} C_VEL
LIN {X 0,Y 334.141,Z 560.55,A -85,B 0,C 180,E1 -14416.532,E2 -14416.532} C_VEL
LIN {X 0,Y 333.761,Z 558.914,A -85,B 0,C 180,E1 -14416.685,E2 -14416.685} C_VEL
LIN {X 0,Y 333.736,Z 558.914,A -85,B 0,C 180,E1 -14419.691,E2 -14419.691} C_VEL
LIN {X 0,Y 333.689,Z 558.92,A -85,B 0,C 180,E1 -14422.279,E2 -14422.279} C_VEL
LIN {X 0,Y 333.733,Z 558.911,A -85,B 0,C 180,E1 -14426.247,E2 -14426.247} C_VEL
LIN {X 0,Y 333.709,Z 558.913,A -85,B 0,C 180,E1 -14428.973,E2 -14428.973} C_VEL
LIN {X 0,Y 333.641,Z 558.913,A -85,B 0,C 180,E1 -14432.588,E2 -14432.588} C_VEL
LIN {X 0,Y 333.674,Z 558.915,A -85,B 0,C 180,E1 -14436.14,E2 -14436.14} C_VEL
LIN {X 0,Y 333.645,Z 558.919,A -85,B 0,C 180,E1 -14439.193,E2 -14439.193} C_VEL
LIN {X 0,Y 333.631,Z 558.923,A -85,B 0,C 180,E1 -14442.501,E2 -14442.501} C_VEL
LIN {X 0,Y 333.621,Z 558.925,A -85,B 0,C 180,E1 -14445.96,E2 -14445.96} C_VEL
LIN {X 0,Y 333.647,Z 558.915,A -85,B 0,C 180,E1 -14449.316,E2 -14449.316} C_VEL
LIN {X 0,Y 333.747,Z 559.118,A -85,B 0,C 180,E1 -14450.628,E2 -14450.628} C_VEL
LIN {X 0,Y 336.542,Z 572.804,A -85,B 0,C 180,E1 -14454.532,E2 -14454.532} C_VEL
LIN {X 0,Y 338.634,Z 583.06,A -85,B 0,C 180,E1 -14457.344,E2 -14457.344} C_VEL
LIN {X 0,Y 336.808,Z 598.729,A -85,B 0,C 180,E1 -14461.32,E2 -14461.32} C_VEL
LIN {X 0,Y 336.335,Z 602.95,A -85,B 0,C 180,E1 -14462.38,E2 -14462.38} C_VEL
LIN {X 0,Y 337.115,Z 608.128,A -85,B 0,C 180,E1 -14462.72,E2 -14462.72} C_VEL
LIN {X 0,Y 339.548,Z 621.101,A -85,B 0,C 180,E1 -14463.558,E2 -14463.558} C_VEL
LIN {X 0,Y 342.786,Z 642.175,A -85,B 0,C 180,E1 -14464.752,E2 -14464.752} C_VEL
LIN {X 0,Y 346.177,Z 683.2,A -85,B 0,C 180,E1 -14466.566,E2 -14466.566} C_VEL
LIN {X 0,Y 344.23,Z 723.794,A -85,B 0,C 180,E1 -14467.77,E2 -14467.77} C_VEL
LIN {X 0,Y 343.01,Z 738.651,A -85,B 0,C 180,E1 -14468.438,E2 -14468.438} C_VEL
LIN {X 0,Y 341.317,Z 753.138,A -85,B 0,C 180,E1 -14469.353,E2 -14469.353} C_VEL
LIN {X 0,Y 339.714,Z 765.3,A -85,B 0,C 180,E1 -14470.357,E2 -14470.357} C_VEL
LIN {X 0,Y 337.807,Z 777.823,A -85,B 0,C 180,E1 -14471.66,E2 -14471.66} C_VEL
LIN {X 0,Y 336.198,Z 789.219,A -85,B 0,C 180,E1 -14473.14,E2 -14473.14} C_VEL
LIN {X 0,Y 334.919,Z 799.486,A -85,B 0,C 180,E1 -14474.799,E2 -14474.799} C_VEL
LIN {X 0,Y 333.847,Z 808.651,A -85,B 0,C 180,E1 -14476.611,E2 -14476.611} C_VEL
LIN {X 0,Y 333.203,Z 816.232,A -85,B 0,C 180,E1 -14478.442,E2 -14478.442} C_VEL
LIN {X 0,Y 332.858,Z 822.389,A -85,B 0,C 180,E1 -14480.276,E2 -14480.276} C_VEL
LIN {X 0,Y 332.838,Z 827.306,A -85,B 0,C 180,E1 -14482.112,E2 -14482.112} C_VEL
LIN {X 0,Y 332.999,Z 831.093,A -85,B 0,C 180,E1 -14483.943,E2 -14483.943} C_VEL
LIN {X 0,Y 333.25,Z 833.3,A -85,B 0,C 180,E1 -14485.162,E2 -14485.162} C_VEL
LIN {X 0,Y 333.28,Z 835.182,A -85,B 0,C 180,E1 -14486.374,E2 -14486.374} C_VEL
LIN {X 0,Y 333.318,Z 836.591,A -85,B 0,C 180,E1 -14487.584,E2 -14487.584} C_VEL
LIN {X 0,Y 333.462,Z 837.518,A -85,B 0,C 180,E1 -14488.793,E2 -14488.793} C_VEL
LIN {X 0,Y 333.666,Z 837.971,A -85,B 0,C 180,E1 -14490.001,E2 -14490.001} C_VEL
LIN {X 0,Y 333.36,Z 837.889,A -85,B 0,C 180,E1 -14491.209,E2 -14491.209} C_VEL
LIN {X 0,Y 333.197,Z 837.38,A -85,B 0,C 180,E1 -14492.418,E2 -14492.418} C_VEL
LIN {X 0,Y 333.13,Z 836.425,A -85,B 0,C 180,E1 -14493.629,E2 -14493.629} C_VEL
LIN {X 0,Y 333.024,Z 834.976,A -85,B 0,C 180,E1 -14494.843,E2 -14494.843} C_VEL
LIN {X 0,Y 332.748,Z 831.422,A -85,B 0,C 180,E1 -14496.928,E2 -14496.928} C_VEL
LIN {X 0,Y 332.695,Z 826.217,A -85,B 0,C 180,E1 -14499.117,E2 -14499.117} C_VEL
LIN {X 0,Y 332.995,Z 819.552,A -85,B 0,C 180,E1 -14501.259,E2 -14501.259} C_VEL
LIN {X 0,Y 333.604,Z 812.424,A -85,B 0,C 180,E1 -14503.09,E2 -14503.09} C_VEL
LIN {X 0,Y 334.603,Z 803.264,A -85,B 0,C 180,E1 -14505.015,E2 -14505.015} C_VEL
LIN {X 0,Y 336.018,Z 793.415,A -85,B 0,C 180,E1 -14506.714,E2 -14506.714} C_VEL
LIN {X 0,Y 337.986,Z 781.937,A -85,B 0,C 180,E1 -14508.332,E2 -14508.332} C_VEL
LIN {X 0,Y 340.007,Z 769.296,A -85,B 0,C 180,E1 -14509.785,E2 -14509.785} C_VEL
LIN {X 0,Y 341.976,Z 757.046,A -85,B 0,C 180,E1 -14510.921,E2 -14510.921} C_VEL
LIN {X 0,Y 344.054,Z 743.024,A -85,B 0,C 180,E1 -14511.968,E2 -14511.968} C_VEL
LIN {X 0,Y 346.082,Z 726.608,A -85,B 0,C 180,E1 -14512.894,E2 -14512.894} C_VEL
LIN {X 0,Y 347.465,Z 711.811,A -85,B 0,C 180,E1 -14513.506,E2 -14513.506} C_VEL
LIN {X 0,Y 349.133,Z 681.734,A -85,B 0,C 180,E1 -14514.464,E2 -14514.464} C_VEL
LIN {X 0,Y 348.512,Z 650.273,A -85,B 0,C 180,E1 -14515.795,E2 -14515.795} C_VEL
LIN {X 0,Y 347.046,Z 630.968,A -85,B 0,C 180,E1 -14516.819,E2 -14516.819} C_VEL
LIN {X 0,Y 344.65,Z 613.049,A -85,B 0,C 180,E1 -14517.993,E2 -14517.993} C_VEL
LIN {X 0,Y 341.911,Z 597.487,A -85,B 0,C 180,E1 -14519.211,E2 -14519.211} C_VEL
LIN {X 0,Y 340.557,Z 590.895,A -85,B 0,C 180,E1 -14519.79,E2 -14519.79} C_VEL
LIN {X 0,Y 339.323,Z 584.815,A -85,B 0,C 180,E1 -14520.355,E2 -14520.355} C_VEL
LIN {X 0,Y 337.825,Z 577.813,A -85,B 0,C 180,E1 -14521.05,E2 -14521.05} C_VEL
LIN {X 0,Y 335.972,Z 570.485,A -85,B 0,C 180,E1 -14521.868,E2 -14521.868} C_VEL
LIN {X 0,Y 335.805,Z 569.47,A -85,B 0,C 180,E1 -14522.043,E2 -14522.043} C_VEL
LIN {X 0,Y 333.722,Z 558.917,A -85,B 0,C 180,E1 -14525.093,E2 -14525.093} C_VEL
LIN {X 0,Y 333.651,Z 558.925,A -85,B 0,C 180,E1 -14529.192,E2 -14529.192} C_VEL
LIN {X 0,Y 333.637,Z 558.923,A -85,B 0,C 180,E1 -14532.5,E2 -14532.5} C_VEL
LIN {X 0,Y 333.601,Z 558.928,A -85,B 0,C 180,E1 -14535.955,E2 -14535.955} C_VEL
LIN {X 0,Y 333.652,Z 558.925,A -85,B 0,C 180,E1 -14539.315,E2 -14539.315} C_VEL
LIN {X 0,Y 333.67,Z 558.922,A -85,B 0,C 180,E1 -14543.168,E2 -14543.168} C_VEL
LIN {X 0,Y 333.679,Z 558.922,A -85,B 0,C 180,E1 -14545.341,E2 -14545.341} C_VEL
LIN {X 0,Y 333.677,Z 559.066,A -85,B 0,C 180,E1 -14548.534,E2 -14548.534} C_VEL
LIN {X 0,Y 334.499,Z 561.51,A -85,B 0,C 180,E1 -14548.869,E2 -14548.869} C_VEL
LIN {X 0,Y 336.553,Z 563.81,A -85,B 0,C 180,E1 -14549.475,E2 -14549.475} C_VEL
LIN {X 0,Y 337.408,Z 564.766,A -85,B 0,C 180,E1 -14549.708,E2 -14549.708} C_VEL
LIN {X 0,Y 339.653,Z 568.189,A -85,B 0,C 180,E1 -14550.35,E2 -14550.35} C_VEL
LIN {X 0,Y 340.697,Z 569.55,A -85,B 0,C 180,E1 -14550.631,E2 -14550.631} C_VEL
LIN {X 0,Y 344.298,Z 575.025,A -85,B 0,C 180,E1 -14551.54,E2 -14551.54} C_VEL
LIN {X 0,Y 348.146,Z 581.225,A -85,B 0,C 180,E1 -14552.442,E2 -14552.442} C_VEL
LIN {X 0,Y 353.191,Z 590.673,A -85,B 0,C 180,E1 -14553.566,E2 -14553.566} C_VEL
LIN {X 0,Y 354.223,Z 593.285,A -85,B 0,C 180,E1 -14553.797,E2 -14553.797} C_VEL
LIN {X 0,Y 353.684,Z 617.391,A -85,B 0,C 180,E1 -14554.516,E2 -14554.516} C_VEL
LIN {X 0,Y 353.403,Z 630.986,A -85,B 0,C 180,E1 -14555.064,E2 -14555.064} C_VEL
LIN {X 0,Y 352.647,Z 645.824,A -85,B 0,C 180,E1 -14555.886,E2 -14555.886} C_VEL
LIN {X 0,Y 351.504,Z 660.114,A -85,B 0,C 180,E1 -14556.938,E2 -14556.938} C_VEL
LIN {X 0,Y 350.061,Z 673.144,A -85,B 0,C 180,E1 -14558.162,E2 -14558.162} C_VEL
LIN {X 0,Y 348.272,Z 685.71,A -85,B 0,C 180,E1 -14559.628,E2 -14559.628} C_VEL
LIN {X 0,Y 346.599,Z 695.917,A -85,B 0,C 180,E1 -14561.068,E2 -14561.068} C_VEL
LIN {X 0,Y 344.711,Z 706.051,A -85,B 0,C 180,E1 -14562.804,E2 -14562.804} C_VEL
LIN {X 0,Y 342.722,Z 715.486,A -85,B 0,C 180,E1 -14564.781,E2 -14564.781} C_VEL
LIN {X 0,Y 340.831,Z 723.69,A -85,B 0,C 180,E1 -14566.889,E2 -14566.889} C_VEL
LIN {X 0,Y 339.432,Z 729.295,A -85,B 0,C 180,E1 -14568.655,E2 -14568.655} C_VEL
LIN {X 0,Y 337.758,Z 735.261,A -85,B 0,C 180,E1 -14571.021,E2 -14571.021} C_VEL
LIN {X 0,Y 336.94,Z 738.726,A -85,B 0,C 180,E1 -14572.81,E2 -14572.81} C_VEL
LIN {X 0,Y 335.876,Z 742.15,A -85,B 0,C 180,E1 -14575.198,E2 -14575.198} C_VEL
LIN {X 0,Y 335.056,Z 744.26,A -85,B 0,C 180,E1 -14577.595,E2 -14577.595} C_VEL
LIN {X 0,Y 334.535,Z 745.098,A -85,B 0,C 180,E1 -14579.999,E2 -14579.999} C_VEL
LIN {X 0,Y 334.104,Z 744.71,A -85,B 0,C 180,E1 -14582.411,E2 -14582.411} C_VEL
LIN {X 0,Y 333.856,Z 743.081,A -85,B 0,C 180,E1 -14584.83,E2 -14584.83} C_VEL
LIN {X 0,Y 334.139,Z 740.137,A -85,B 0,C 180,E1 -14587.249,E2 -14587.249} C_VEL
LIN {X 0,Y 334.317,Z 735.888,A -85,B 0,C 180,E1 -14589.681,E2 -14589.681} C_VEL
LIN {X 0,Y 334.714,Z 730.182,A -85,B 0,C 180,E1 -14592.12,E2 -14592.12} C_VEL
LIN {X 0,Y 335.146,Z 724.801,A -85,B 0,C 180,E1 -14593.954,E2 -14593.954} C_VEL
LIN {X 0,Y 335.861,Z 717.239,A -85,B 0,C 180,E1 -14596.096,E2 -14596.096} C_VEL
LIN {X 0,Y 336.818,Z 708.032,A -85,B 0,C 180,E1 -14598.239,E2 -14598.239} C_VEL
LIN {X 0,Y 337.821,Z 698.538,A -85,B 0,C 180,E1 -14600.075,E2 -14600.075} C_VEL
LIN {X 0,Y 338.952,Z 687.188,A -85,B 0,C 180,E1 -14601.914,E2 -14601.914} C_VEL
LIN {X 0,Y 340.091,Z 674.624,A -85,B 0,C 180,E1 -14603.602,E2 -14603.602} C_VEL
LIN {X 0,Y 341.108,Z 662.329,A -85,B 0,C 180,E1 -14604.966,E2 -14604.966} C_VEL
LIN {X 0,Y 342.123,Z 648.633,A -85,B 0,C 180,E1 -14606.209,E2 -14606.209} C_VEL
LIN {X 0,Y 342.991,Z 633.588,A -85,B 0,C 180,E1 -14607.288,E2 -14607.288} C_VEL
LIN {X 0,Y 343.652,Z 618.449,A -85,B 0,C 180,E1 -14608.112,E2 -14608.112} C_VEL
LIN {X 0,Y 343.919,Z 602.825,A -85,B 0,C 180,E1 -14608.719,E2 -14608.719} C_VEL
LIN {X 0,Y 344.092,Z 587.16,A -85,B 0,C 180,E1 -14609.166,E2 -14609.166} C_VEL
LIN {X 0,Y 333.686,Z 558.918,A -85,B 0,C 180,E1 -14610.558,E2 -14610.558} C_VEL
LIN {X 0,Y 333.686,Z 558.917,A -85,B 0,C 180,E1 -14614.773,E2 -14614.773} C_VEL
LIN {X 0,Y 333.653,Z 558.921,A -85,B 0,C 180,E1 -14617.65,E2 -14617.65} C_VEL
LIN {X 0,Y 333.647,Z 558.922,A -85,B 0,C 180,E1 -14620.767,E2 -14620.767} C_VEL
LIN {X 0,Y 333.594,Z 558.933,A -85,B 0,C 180,E1 -14624.25,E2 -14624.25} C_VEL
LIN {X 0,Y 333.642,Z 558.922,A -85,B 0,C 180,E1 -14627.618,E2 -14627.618} C_VEL
LIN {X 0,Y 333.654,Z 558.92,A -85,B 0,C 180,E1 -14631.201,E2 -14631.201} C_VEL
LIN {X 0,Y 333.677,Z 558.918,A -85,B 0,C 180,E1 -14633.86,E2 -14633.86} C_VEL
LIN {X 0,Y 333.643,Z 558.921,A -85,B 0,C 180,E1 -14637.412,E2 -14637.412} C_VEL
LIN {X 0,Y 333.689,Z 558.918,A -85,B 0,C 180,E1 -14641.025,E2 -14641.025} C_VEL
LIN {X 0,Y 333.734,Z 558.91,A -85,B 0,C 180,E1 -14643.753,E2 -14643.753} C_VEL
LIN {X 0,Y 333.718,Z 558.912,A -85,B 0,C 180,E1 -14647.913,E2 -14647.913} C_VEL
LIN {X 0,Y 333.792,Z 558.903,A -85,B 0,C 180,E1 -14651.589,E2 -14651.589} C_VEL
LIN {X 0,Y 333.807,Z 558.901,A -85,B 0,C 180,E1 -14655.576,E2 -14655.576} C_VEL
LIN {X 0,Y 333.832,Z 558.903,A -85,B 0,C 180,E1 -14659.077,E2 -14659.077} C_VEL
LIN {X 0,Y 334.024,Z 558.877,A -85,B 0,C 180,E1 -14662.747,E2 -14662.747} C_VEL
LIN {X 0,Y 333.81,Z 558.906,A -85,B 0,C 180,E1 -14665.168,E2 -14665.168} C_VEL
LIN {X 0,Y 334.105,Z 558.865,A -85,B 0,C 180,E1 -14667.588,E2 -14667.588} C_VEL
LIN {X 0,Y 334.245,Z 558.846,A -85,B 0,C 180,E1 -14669.999,E2 -14669.999} C_VEL
LIN {X 0,Y 334.105,Z 558.864,A -85,B 0,C 180,E1 -14672.41,E2 -14672.41} C_VEL
LIN {X 0,Y 334.021,Z 558.88,A -85,B 0,C 180,E1 -14677.252,E2 -14677.252} C_VEL
LIN {X 0,Y 333.834,Z 558.9,A -85,B 0,C 180,E1 -14680.921,E2 -14680.921} C_VEL
LIN {X 0,Y 333.805,Z 558.901,A -85,B 0,C 180,E1 -14684.634,E2 -14684.634} C_VEL
LIN {X 0,Y 333.792,Z 558.903,A -85,B 0,C 180,E1 -14688.654,E2 -14688.654} C_VEL
LIN {X 0,Y 333.688,Z 558.916,A -85,B 0,C 180,E1 -14692.278,E2 -14692.278} C_VEL
LIN {X 0,Y 333.732,Z 558.911,A -85,B 0,C 180,E1 -14696.246,E2 -14696.246} C_VEL
LIN {X 0,Y 333.708,Z 558.914,A -85,B 0,C 180,E1 -14698.971,E2 -14698.971} C_VEL
LIN {X 0,Y 333.647,Z 558.921,A -85,B 0,C 180,E1 -14702.589,E2 -14702.589} C_VEL
LIN {X 0,Y 333.672,Z 558.921,A -85,B 0,C 180,E1 -14706.138,E2 -14706.138} C_VEL
LIN {X 0,Y 333.667,Z 558.919,A -85,B 0,C 180,E1 -14709.188,E2 -14709.188} C_VEL
LIN {X 0,Y 333.67,Z 558.919,A -85,B 0,C 180,E1 -14712.508,E2 -14712.508} C_VEL
LIN {X 0,Y 333.718,Z 558.918,A -85,B 0,C 180,E1 -14715.976,E2 -14715.976} C_VEL
LIN {X 0,Y 333.696,Z 558.915,A -85,B 0,C 180,E1 -14719.304,E2 -14719.304} C_VEL
LIN {X 0,Y 333.708,Z 558.919,A -85,B 0,C 180,E1 -14722.056,E2 -14722.056} C_VEL
LIN {X 0,Y 337.879,Z 570.527,A -85,B 0,C 180,E1 -14722.641,E2 -14722.641} C_VEL
LIN {X 0,Y 342.958,Z 584.006,A -85,B 0,C 180,E1 -14723.267,E2 -14723.267} C_VEL
LIN {X 0,Y 342.597,Z 599.34,A -85,B 0,C 180,E1 -14723.654,E2 -14723.654} C_VEL
LIN {X 0,Y 341.866,Z 605.159,A -85,B 0,C 180,E1 -14723.771,E2 -14723.771} C_VEL
LIN {X 0,Y 336.059,Z 624.032,A -85,B 0,C 180,E1 -14724.048,E2 -14724.048} C_VEL
LIN {X 0,Y 335.333,Z 629.768,A -85,B 0,C 180,E1 -14724.251,E2 -14724.251} C_VEL
LIN {X 0,Y 334.781,Z 644.364,A -85,B 0,C 180,E1 -14725.017,E2 -14725.017} C_VEL
LIN {X 0,Y 334.015,Z 658.329,A -85,B 0,C 180,E1 -14726.021,E2 -14726.021} C_VEL
LIN {X 0,Y 333.168,Z 670.617,A -85,B 0,C 180,E1 -14727.147,E2 -14727.147} C_VEL
LIN {X 0,Y 332.101,Z 683.355,A -85,B 0,C 180,E1 -14728.593,E2 -14728.593} C_VEL
LIN {X 0,Y 331.041,Z 694.315,A -85,B 0,C 180,E1 -14730.131,E2 -14730.131} C_VEL
LIN {X 0,Y 330.15,Z 703.765,A -85,B 0,C 180,E1 -14731.73,E2 -14731.73} C_VEL
LIN {X 0,Y 329.174,Z 713.51,A -85,B 0,C 180,E1 -14733.728,E2 -14733.728} C_VEL
LIN {X 0,Y 328.352,Z 721.259,A -85,B 0,C 180,E1 -14735.669,E2 -14735.669} C_VEL
LIN {X 0,Y 327.668,Z 728.593,A -85,B 0,C 180,E1 -14737.955,E2 -14737.955} C_VEL
LIN {X 0,Y 327.225,Z 733.549,A -85,B 0,C 180,E1 -14739.902,E2 -14739.902} C_VEL
LIN {X 0,Y 326.932,Z 737.417,A -85,B 0,C 180,E1 -14741.839,E2 -14741.839} C_VEL
LIN {X 0,Y 326.737,Z 740.29,A -85,B 0,C 180,E1 -14743.763,E2 -14743.763} C_VEL
LIN {X 0,Y 326.738,Z 742.08,A -85,B 0,C 180,E1 -14745.447,E2 -14745.447} C_VEL
LIN {X 0,Y 326.868,Z 743.403,A -85,B 0,C 180,E1 -14747.584,E2 -14747.584} C_VEL
LIN {X 0,Y 327.242,Z 743.582,A -85,B 0,C 180,E1 -14750.107,E2 -14750.107} C_VEL
LIN {X 0,Y 327.786,Z 742.324,A -85,B 0,C 180,E1 -14752.609,E2 -14752.609} C_VEL
LIN {X 0,Y 328.239,Z 741.119,A -85,B 0,C 180,E1 -14753.855,E2 -14753.855} C_VEL
LIN {X 0,Y 329.237,Z 737.563,A -85,B 0,C 180,E1 -14756.329,E2 -14756.329} C_VEL
LIN {X 0,Y 330.514,Z 732.429,A -85,B 0,C 180,E1 -14758.782,E2 -14758.782} C_VEL
LIN {X 0,Y 331.689,Z 727.38,A -85,B 0,C 180,E1 -14760.608,E2 -14760.608} C_VEL
LIN {X 0,Y 333.194,Z 720.093,A -85,B 0,C 180,E1 -14762.721,E2 -14762.721} C_VEL
LIN {X 0,Y 334.878,Z 712.265,A -85,B 0,C 180,E1 -14764.514,E2 -14764.514} C_VEL
LIN {X 0,Y 336.519,Z 702.859,A -85,B 0,C 180,E1 -14766.295,E2 -14766.295} C_VEL
LIN {X 0,Y 338.24,Z 692.269,A -85,B 0,C 180,E1 -14767.913,E2 -14767.913} C_VEL
LIN {X 0,Y 339.887,Z 680.411,A -85,B 0,C 180,E1 -14769.372,E2 -14769.372} C_VEL
LIN {X 0,Y 341.245,Z 668.473,A -85,B 0,C 180,E1 -14770.532,E2 -14770.532} C_VEL
LIN {X 0,Y 342.278,Z 655.483,A -85,B 0,C 180,E1 -14771.549,E2 -14771.549} C_VEL
LIN {X 0,Y 343.02,Z 641.846,A -85,B 0,C 180,E1 -14772.352,E2 -14772.352} C_VEL
LIN {X 0,Y 343.339,Z 627.282,A -85,B 0,C 180,E1 -14772.941,E2 -14772.941} C_VEL
LIN {X 0,Y 344.292,Z 594.307,A -85,B 0,C 180,E1 -14773.876,E2 -14773.876} C_VEL
LIN {X 0,Y 344.239,Z 590.904,A -85,B 0,C 180,E1 -14773.992,E2 -14773.992} C_VEL
LIN {X 0,Y 338.089,Z 578.758,A -85,B 0,C 180,E1 -14775.244,E2 -14775.244} C_VEL
LIN {X 0,Y 331.758,Z 568.367,A -85,B 0,C 180,E1 -14776.603,E2 -14776.603} C_VEL
LIN {X 0,Y 329.684,Z 565.143,A -85,B 0,C 180,E1 -14777.073,E2 -14777.073} C_VEL
LIN {X 0,Y 327.292,Z 561.83,A -85,B 0,C 180,E1 -14777.627,E2 -14777.627} C_VEL
LIN {X 0,Y 326.715,Z 559.79,A -85,B 0,C 180,E1 -14777.851,E2 -14777.851} C_VEL
LIN {X 0,Y 326.644,Z 559.796,A -85,B 0,C 180,E1 -14781.455,E2 -14781.455} C_VEL
LIN {X 0,Y 326.687,Z 559.787,A -85,B 0,C 180,E1 -14785.485,E2 -14785.485} C_VEL
LIN {X 0,Y 326.658,Z 559.786,A -85,B 0,C 180,E1 -14789.66,E2 -14789.66} C_VEL
LIN {X 0,Y 326.605,Z 559.792,A -85,B 0,C 180,E1 -14794.02,E2 -14794.02} C_VEL
LIN {X 0,Y 326.626,Z 559.791,A -85,B 0,C 180,E1 -14797.24,E2 -14797.24} C_VEL
LIN {X 0,Y 326.577,Z 559.805,A -85,B 0,C 180,E1 -14801.132,E2 -14801.132} C_VEL
LIN {X 0,Y 326.555,Z 559.807,A -85,B 0,C 180,E1 -14804.749,E2 -14804.749} C_VEL
LIN {X 0,Y 326.576,Z 559.798,A -85,B 0,C 180,E1 -14808.155,E2 -14808.155} C_VEL
LIN {X 0,Y 326.683,Z 559.915,A -85,B 0,C 180,E1 -14810.391,E2 -14810.391} C_VEL
LIN {X 0,Y 329.567,Z 574.13,A -85,B 0,C 180,E1 -14814.537,E2 -14814.537} C_VEL
LIN {X 0,Y 331.602,Z 583.971,A -85,B 0,C 180,E1 -14817.287,E2 -14817.287} C_VEL
LIN {X 0,Y 329.735,Z 599.242,A -85,B 0,C 180,E1 -14821.251,E2 -14821.251} C_VEL
LIN {X 0,Y 330.411,Z 604.096,A -85,B 0,C 180,E1 -14821.573,E2 -14821.573} C_VEL
LIN {X 0,Y 331.041,Z 606.939,A -85,B 0,C 180,E1 -14821.791,E2 -14821.791} C_VEL
LIN {X 0,Y 333.444,Z 620.104,A -85,B 0,C 180,E1 -14822.689,E2 -14822.689} C_VEL
LIN {X 0,Y 336.475,Z 639.549,A -85,B 0,C 180,E1 -14823.876,E2 -14823.876} C_VEL
LIN {X 0,Y 337.614,Z 651.748,A -85,B 0,C 180,E1 -14824.485,E2 -14824.485} C_VEL
LIN {X 0,Y 340.155,Z 683.679,A -85,B 0,C 180,E1 -14825.943,E2 -14825.943} C_VEL
LIN {X 0,Y 338.196,Z 721.897,A -85,B 0,C 180,E1 -14827.109,E2 -14827.109} C_VEL
LIN {X 0,Y 336.867,Z 736.694,A -85,B 0,C 180,E1 -14827.782,E2 -14827.782} C_VEL
LIN {X 0,Y 335.224,Z 750.22,A -85,B 0,C 180,E1 -14828.638,E2 -14828.638} C_VEL
LIN {X 0,Y 333.313,Z 764.266,A -85,B 0,C 180,E1 -14829.802,E2 -14829.802} C_VEL
LIN {X 0,Y 331.527,Z 775.444,A -85,B 0,C 180,E1 -14830.979,E2 -14830.979} C_VEL
LIN {X 0,Y 329.71,Z 786.945,A -85,B 0,C 180,E1 -14832.478,E2 -14832.478} C_VEL
LIN {X 0,Y 328.244,Z 797.392,A -85,B 0,C 180,E1 -14834.159,E2 -14834.159} C_VEL
LIN {X 0,Y 327.097,Z 806.724,A -85,B 0,C 180,E1 -14836.013,E2 -14836.013} C_VEL
LIN {X 0,Y 326.259,Z 814.398,A -85,B 0,C 180,E1 -14837.877,E2 -14837.877} C_VEL
LIN {X 0,Y 325.789,Z 821.606,A -85,B 0,C 180,E1 -14840.063,E2 -14840.063} C_VEL
LIN {X 0,Y 325.756,Z 826.457,A -85,B 0,C 180,E1 -14841.939,E2 -14841.939} C_VEL
LIN {X 0,Y 325.916,Z 830.186,A -85,B 0,C 180,E1 -14843.811,E2 -14843.811} C_VEL
LIN {X 0,Y 326.262,Z 833.885,A -85,B 0,C 180,E1 -14846.296,E2 -14846.296} C_VEL
LIN {X 0,Y 326.334,Z 835.347,A -85,B 0,C 180,E1 -14847.532,E2 -14847.532} C_VEL
LIN {X 0,Y 326.448,Z 836.343,A -85,B 0,C 180,E1 -14848.767,E2 -14848.767} C_VEL
LIN {X 0,Y 326.654,Z 836.847,A -85,B 0,C 180,E1 -14850.001,E2 -14850.001} C_VEL
LIN {X 0,Y 326.352,Z 836.805,A -85,B 0,C 180,E1 -14851.235,E2 -14851.235} C_VEL
LIN {X 0,Y 326.159,Z 836.327,A -85,B 0,C 180,E1 -14852.471,E2 -14852.471} C_VEL
LIN {X 0,Y 326.082,Z 835.42,A -85,B 0,C 180,E1 -14853.708,E2 -14853.708} C_VEL
LIN {X 0,Y 325.94,Z 834.04,A -85,B 0,C 180,E1 -14854.949,E2 -14854.949} C_VEL
LIN {X 0,Y 325.69,Z 830.815,A -85,B 0,C 180,E1 -14856.959,E2 -14856.959} C_VEL
LIN {X 0,Y 325.616,Z 825.468,A -85,B 0,C 180,E1 -14859.317,E2 -14859.317} C_VEL
LIN {X 0,Y 325.982,Z 818.917,A -85,B 0,C 180,E1 -14861.504,E2 -14861.504} C_VEL
LIN {X 0,Y 326.769,Z 810.65,A -85,B 0,C 180,E1 -14863.686,E2 -14863.686} C_VEL
LIN {X 0,Y 327.592,Z 803.669,A -85,B 0,C 180,E1 -14865.205,E2 -14865.205} C_VEL
LIN {X 0,Y 329.226,Z 793.39,A -85,B 0,C 180,E1 -14867.07,E2 -14867.07} C_VEL
LIN {X 0,Y 331.441,Z 781.076,A -85,B 0,C 180,E1 -14868.867,E2 -14868.867} C_VEL
LIN {X 0,Y 333.577,Z 768.671,A -85,B 0,C 180,E1 -14870.343,E2 -14870.343} C_VEL
LIN {X 0,Y 335.987,Z 754.991,A -85,B 0,C 180,E1 -14871.634,E2 -14871.634} C_VEL
LIN {X 0,Y 338.196,Z 740.965,A -85,B 0,C 180,E1 -14872.691,E2 -14872.691} C_VEL
LIN {X 0,Y 340.329,Z 724.675,A -85,B 0,C 180,E1 -14873.626,E2 -14873.626} C_VEL
LIN {X 0,Y 341.84,Z 709.132,A -85,B 0,C 180,E1 -14874.28,E2 -14874.28} C_VEL
LIN {X 0,Y 343.425,Z 682.005,A -85,B 0,C 180,E1 -14875.18,E2 -14875.18} C_VEL
LIN {X 0,Y 343.045,Z 651.918,A -85,B 0,C 180,E1 -14876.498,E2 -14876.498} C_VEL
LIN {X 0,Y 341.822,Z 633.25,A -85,B 0,C 180,E1 -14877.518,E2 -14877.518} C_VEL
LIN {X 0,Y 339.655,Z 615.779,A -85,B 0,C 180,E1 -14878.71,E2 -14878.71} C_VEL
LIN {X 0,Y 337.321,Z 601.151,A -85,B 0,C 180,E1 -14879.884,E2 -14879.884} C_VEL
LIN {X 0,Y 334.861,Z 588.237,A -85,B 0,C 180,E1 -14881.094,E2 -14881.094} C_VEL
LIN {X 0,Y 333.337,Z 580.903,A -85,B 0,C 180,E1 -14881.862,E2 -14881.862} C_VEL
LIN {X 0,Y 331.708,Z 573.989,A -85,B 0,C 180,E1 -14882.688,E2 -14882.688} C_VEL
LIN {X 0,Y 328.25,Z 565.736,A -85,B 0,C 180,E1 -14884.181,E2 -14884.181} C_VEL
LIN {X 0,Y 327.116,Z 561.851,A -85,B 0,C 180,E1 -14884.811,E2 -14884.811} C_VEL
LIN {X 0,Y 326.695,Z 559.792,A -85,B 0,C 180,E1 -14885.51,E2 -14885.51} C_VEL
LIN {X 0,Y 326.616,Z 559.801,A -85,B 0,C 180,E1 -14889.227,E2 -14889.227} C_VEL
LIN {X 0,Y 326.58,Z 559.806,A -85,B 0,C 180,E1 -14892.972,E2 -14892.972} C_VEL
LIN {X 0,Y 326.581,Z 559.805,A -85,B 0,C 180,E1 -14897.028,E2 -14897.028} C_VEL
LIN {X 0,Y 326.616,Z 559.798,A -85,B 0,C 180,E1 -14900.773,E2 -14900.773} C_VEL
LIN {X 0,Y 326.617,Z 559.798,A -85,B 0,C 180,E1 -14904.48,E2 -14904.48} C_VEL
LIN {X 0,Y 326.634,Z 559.997,A -85,B 0,C 180,E1 -14906.63,E2 -14906.63} C_VEL
LIN {X 0,Y 327.476,Z 562.417,A -85,B 0,C 180,E1 -14907.037,E2 -14907.037} C_VEL
LIN {X 0,Y 329.55,Z 564.732,A -85,B 0,C 180,E1 -14907.781,E2 -14907.781} C_VEL
LIN {X 0,Y 330.54,Z 565.588,A -85,B 0,C 180,E1 -14908.098,E2 -14908.098} C_VEL
LIN {X 0,Y 332.408,Z 568.737,A -85,B 0,C 180,E1 -14908.743,E2 -14908.743} C_VEL
LIN {X 0,Y 334.1,Z 570.629,A -85,B 0,C 180,E1 -14909.258,E2 -14909.258} C_VEL
LIN {X 0,Y 336.816,Z 574.437,A -85,B 0,C 180,E1 -14910.041,E2 -14910.041} C_VEL
LIN {X 0,Y 342.341,Z 583.128,A -85,B 0,C 180,E1 -14911.51,E2 -14911.51} C_VEL
LIN {X 0,Y 346.959,Z 591.588,A -85,B 0,C 180,E1 -14912.628,E2 -14912.628} C_VEL
LIN {X 0,Y 348.833,Z 595.639,A -85,B 0,C 180,E1 -14913.076,E2 -14913.076} C_VEL
LIN {X 0,Y 348.229,Z 620.937,A -85,B 0,C 180,E1 -14913.879,E2 -14913.879} C_VEL
LIN {X 0,Y 347.825,Z 635.363,A -85,B 0,C 180,E1 -14914.506,E2 -14914.506} C_VEL
LIN {X 0,Y 347.054,Z 648.299,A -85,B 0,C 180,E1 -14915.272,E2 -14915.272} C_VEL
LIN {X 0,Y 345.796,Z 662.001,A -85,B 0,C 180,E1 -14916.319,E2 -14916.319} C_VEL
LIN {X 0,Y 344.336,Z 674.406,A -85,B 0,C 180,E1 -14917.499,E2 -14917.499} C_VEL
LIN {X 0,Y 342.477,Z 686.761,A -85,B 0,C 180,E1 -14918.953,E2 -14918.953} C_VEL
LIN {X 0,Y 340.667,Z 696.94,A -85,B 0,C 180,E1 -14920.412,E2 -14920.412} C_VEL
LIN {X 0,Y 338.674,Z 707.112,A -85,B 0,C 180,E1 -14922.176,E2 -14922.176} C_VEL
LIN {X 0,Y 336.838,Z 715.427,A -85,B 0,C 180,E1 -14923.902,E2 -14923.902} C_VEL
LIN {X 0,Y 335.025,Z 722.725,A -85,B 0,C 180,E1 -14925.73,E2 -14925.73} C_VEL
LIN {X 0,Y 333.229,Z 729.555,A -85,B 0,C 180,E1 -14927.824,E2 -14927.824} C_VEL
LIN {X 0,Y 331.399,Z 735.787,A -85,B 0,C 180,E1 -14930.232,E2 -14930.232} C_VEL
LIN {X 0,Y 330.424,Z 739.343,A -85,B 0,C 180,E1 -14932.053,E2 -14932.053} C_VEL
LIN {X 0,Y 329.503,Z 742.171,A -85,B 0,C 180,E1 -14933.877,E2 -14933.877} C_VEL
LIN {X 0,Y 328.428,Z 744.781,A -85,B 0,C 180,E1 -14936.319,E2 -14936.319} C_VEL
LIN {X 0,Y 327.776,Z 746.103,A -85,B 0,C 180,E1 -14938.771,E2 -14938.771} C_VEL
LIN {X 0,Y 327.322,Z 746.179,A -85,B 0,C 180,E1 -14941.23,E2 -14941.23} C_VEL
LIN {X 0,Y 326.997,Z 745.016,A -85,B 0,C 180,E1 -14943.696,E2 -14943.696} C_VEL
LIN {X 0,Y 327.009,Z 742.58,A -85,B 0,C 180,E1 -14946.168,E2 -14946.168} C_VEL
LIN {X 0,Y 327.139,Z 738.837,A -85,B 0,C 180,E1 -14948.649,E2 -14948.649} C_VEL
LIN {X 0,Y 327.472,Z 733.674,A -85,B 0,C 180,E1 -14951.136,E2 -14951.136} C_VEL
LIN {X 0,Y 327.974,Z 726.937,A -85,B 0,C 180,E1 -14953.633,E2 -14953.633} C_VEL
LIN {X 0,Y 328.675,Z 719.669,A -85,B 0,C 180,E1 -14955.796,E2 -14955.796} C_VEL
LIN {X 0,Y 329.511,Z 712.021,A -85,B 0,C 180,E1 -14957.693,E2 -14957.693} C_VEL
LIN {X 0,Y 330.455,Z 703.059,A -85,B 0,C 180,E1 -14959.57,E2 -14959.57} C_VEL
LIN {X 0,Y 331.571,Z 692.355,A -85,B 0,C 180,E1 -14961.446,E2 -14961.446} C_VEL
LIN {X 0,Y 332.692,Z 680.566,A -85,B 0,C 180,E1 -14963.169,E2 -14963.169} C_VEL
LIN {X 0,Y 333.876,Z 667.63,A -85,B 0,C 180,E1 -14964.731,E2 -14964.731} C_VEL
LIN {X 0,Y 334.863,Z 654.733,A -85,B 0,C 180,E1 -14966.015,E2 -14966.015} C_VEL
LIN {X 0,Y 335.777,Z 640.406,A -85,B 0,C 180,E1 -14967.164,E2 -14967.164} C_VEL
LIN {X 0,Y 336.548,Z 625.174,A -85,B 0,C 180,E1 -14968.109,E2 -14968.109} C_VEL
LIN {X 0,Y 337.034,Z 610.243,A -85,B 0,C 180,E1 -14968.79,E2 -14968.79} C_VEL
LIN {X 0,Y 337.129,Z 588.303,A -85,B 0,C 180,E1 -14969.474,E2 -14969.474} C_VEL
LIN {X 0,Y 326.631,Z 559.824,A -85,B 0,C 180,E1 -14970.91,E2 -14970.91} C_VEL
LIN {X 0,Y 326.608,Z 559.803,A -85,B 0,C 180,E1 -14974.019,E2 -14974.019} C_VEL
LIN {X 0,Y 326.628,Z 559.795,A -85,B 0,C 180,E1 -14977.238,E2 -14977.238} C_VEL
LIN {X 0,Y 326.578,Z 559.801,A -85,B 0,C 180,E1 -14981.13,E2 -14981.13} C_VEL
LIN {X 0,Y 326.528,Z 559.81,A -85,B 0,C 180,E1 -14984.742,E2 -14984.742} C_VEL
LIN {X 0,Y 326.576,Z 559.805,A -85,B 0,C 180,E1 -14988.153,E2 -14988.153} C_VEL
LIN {X 0,Y 326.624,Z 559.796,A -85,B 0,C 180,E1 -14991.391,E2 -14991.391} C_VEL
LIN {X 0,Y 326.62,Z 559.799,A -85,B 0,C 180,E1 -14994.85,E2 -14994.85} C_VEL
LIN {X 0,Y 326.607,Z 559.798,A -85,B 0,C 180,E1 -14997.455,E2 -14997.455} C_VEL
LIN {X 0,Y 326.647,Z 559.796,A -85,B 0,C 180,E1 -15000.339,E2 -15000.339} C_VEL
LIN {X 0,Y 326.689,Z 559.792,A -85,B 0,C 180,E1 -15004.515,E2 -15004.515} C_VEL
LIN {X 0,Y 326.647,Z 559.797,A -85,B 0,C 180,E1 -15008.545,E2 -15008.545} C_VEL
LIN {X 0,Y 326.743,Z 559.783,A -85,B 0,C 180,E1 -15011.177,E2 -15011.177} C_VEL
LIN {X 0,Y 326.761,Z 559.78,A -85,B 0,C 180,E1 -15015.432,E2 -15015.432} C_VEL
LIN {X 0,Y 326.768,Z 559.783,A -85,B 0,C 180,E1 -15018.838,E2 -15018.838} C_VEL
LIN {X 0,Y 326.978,Z 559.754,A -85,B 0,C 180,E1 -15022.59,E2 -15022.59} C_VEL
LIN {X 0,Y 326.777,Z 559.783,A -85,B 0,C 180,E1 -15025.064,E2 -15025.064} C_VEL
LIN {X 0,Y 327.046,Z 559.745,A -85,B 0,C 180,E1 -15027.536,E2 -15027.536} C_VEL
LIN {X 0,Y 327.197,Z 559.724,A -85,B 0,C 180,E1 -15029.999,E2 -15029.999} C_VEL
LIN {X 0,Y 327.046,Z 559.744,A -85,B 0,C 180,E1 -15032.463,E2 -15032.463} C_VEL
LIN {X 0,Y 326.992,Z 559.75,A -85,B 0,C 180,E1 -15036.168,E2 -15036.168} C_VEL
LIN {X 0,Y 326.911,Z 559.761,A -85,B 0,C 180,E1 -15038.654,E2 -15038.654} C_VEL
LIN {X 0,Y 326.735,Z 559.782,A -85,B 0,C 180,E1 -15042.42,E2 -15042.42} C_VEL
LIN {X 0,Y 326.75,Z 559.782,A -85,B 0,C 180,E1 -15044.957,E2 -15044.957} C_VEL
LIN {X 0,Y 326.728,Z 559.783,A -85,B 0,C 180,E1 -15048.837,E2 -15048.837} C_VEL
LIN {X 0,Y 326.617,Z 559.797,A -85,B 0,C 180,E1 -15052.787,E2 -15052.787} C_VEL
LIN {X 0,Y 326.686,Z 559.793,A -85,B 0,C 180,E1 -15055.483,E2 -15055.483} C_VEL
LIN {X 0,Y 326.657,Z 559.798,A -85,B 0,C 180,E1 -15059.658,E2 -15059.658} C_VEL
LIN {X 0,Y 326.618,Z 559.797,A -85,B 0,C 180,E1 -15062.947,E2 -15062.947} C_VEL
LIN {X 0,Y 326.628,Z 559.795,A -85,B 0,C 180,E1 -15067.046,E2 -15067.046} C_VEL
LIN {X 0,Y 326.599,Z 559.802,A -85,B 0,C 180,E1 -15070.207,E2 -15070.207} C_VEL
LIN {X 0,Y 326.618,Z 559.798,A -85,B 0,C 180,E1 -15073.515,E2 -15073.515} C_VEL
LIN {X 0,Y 326.643,Z 559.793,A -85,B 0,C 180,E1 -15077.014,E2 -15077.014} C_VEL
LIN {X 0,Y 326.64,Z 559.794,A -85,B 0,C 180,E1 -15080.765,E2 -15080.765} C_VEL
LIN {X 0,Y 326.649,Z 559.795,A -85,B 0,C 180,E1 -15081.697,E2 -15081.697} C_VEL
LIN {X 0,Y 336.131,Z 585.437,A -85,B 0,C 180,E1 -15082.949,E2 -15082.949} C_VEL
LIN {X 0,Y 335.438,Z 622.575,A -85,B 0,C 180,E1 -15083.966,E2 -15083.966} C_VEL
LIN {X 0,Y 335.333,Z 629.768,A -85,B 0,C 180,E1 -15084.251,E2 -15084.251} C_VEL
LIN {X 0,Y 334.502,Z 635.475,A -85,B 0,C 180,E1 -15084.478,E2 -15084.478} C_VEL
LIN {X 0,Y 331.319,Z 644.638,A -85,B 0,C 180,E1 -15084.849,E2 -15084.849} C_VEL
LIN {X 0,Y 328.076,Z 653.583,A -85,B 0,C 180,E1 -15085.333,E2 -15085.333} C_VEL
LIN {X 0,Y 327.158,Z 658.945,A -85,B 0,C 180,E1 -15085.733,E2 -15085.733} C_VEL
LIN {X 0,Y 326.269,Z 671.562,A -85,B 0,C 180,E1 -15086.908,E2 -15086.908} C_VEL
LIN {X 0,Y 325.284,Z 683.011,A -85,B 0,C 180,E1 -15088.222,E2 -15088.222} C_VEL
LIN {X 0,Y 324.204,Z 693.907,A -85,B 0,C 180,E1 -15089.735,E2 -15089.735} C_VEL
LIN {X 0,Y 323.237,Z 703.915,A -85,B 0,C 180,E1 -15091.424,E2 -15091.424} C_VEL
LIN {X 0,Y 322.237,Z 713.56,A -85,B 0,C 180,E1 -15093.405,E2 -15093.405} C_VEL
LIN {X 0,Y 321.376,Z 721.717,A -85,B 0,C 180,E1 -15095.45,E2 -15095.45} C_VEL
LIN {X 0,Y 320.731,Z 728.397,A -85,B 0,C 180,E1 -15097.507,E2 -15097.507} C_VEL
LIN {X 0,Y 320.258,Z 733.483,A -85,B 0,C 180,E1 -15099.445,E2 -15099.445} C_VEL
LIN {X 0,Y 319.927,Z 737.64,A -85,B 0,C 180,E1 -15101.439,E2 -15101.439} C_VEL
LIN {X 0,Y 319.71,Z 740.76,A -85,B 0,C 180,E1 -15103.396,E2 -15103.396} C_VEL
LIN {X 0,Y 319.741,Z 743.514,A -85,B 0,C 180,E1 -15106.009,E2 -15106.009} C_VEL
LIN {X 0,Y 319.97,Z 744.757,A -85,B 0,C 180,E1 -15108.599,E2 -15108.599} C_VEL
LIN {X 0,Y 320.445,Z 744.458,A -85,B 0,C 180,E1 -15111.169,E2 -15111.169} C_VEL
LIN {X 0,Y 321.196,Z 742.711,A -85,B 0,C 180,E1 -15113.72,E2 -15113.72} C_VEL
LIN {X 0,Y 322.255,Z 739.484,A -85,B 0,C 180,E1 -15116.249,E2 -15116.249} C_VEL
LIN {X 0,Y 323.403,Z 735.341,A -85,B 0,C 180,E1 -15118.437,E2 -15118.437} C_VEL
LIN {X 0,Y 324.823,Z 729.796,A -85,B 0,C 180,E1 -15120.62,E2 -15120.62} C_VEL
LIN {X 0,Y 326.38,Z 722.854,A -85,B 0,C 180,E1 -15122.778,E2 -15122.778} C_VEL
LIN {X 0,Y 328.063,Z 715.43,A -85,B 0,C 180,E1 -15124.608,E2 -15124.608} C_VEL
LIN {X 0,Y 329.884,Z 706.418,A -85,B 0,C 180,E1 -15126.422,E2 -15126.422} C_VEL
LIN {X 0,Y 331.581,Z 696.388,A -85,B 0,C 180,E1 -15128.073,E2 -15128.073} C_VEL
LIN {X 0,Y 333.361,Z 685.176,A -85,B 0,C 180,E1 -15129.557,E2 -15129.557} C_VEL
LIN {X 0,Y 334.804,Z 674.223,A -85,B 0,C 180,E1 -15130.737,E2 -15130.737} C_VEL
LIN {X 0,Y 335.974,Z 662.41,A -85,B 0,C 180,E1 -15131.769,E2 -15131.769} C_VEL
LIN {X 0,Y 336.853,Z 649.473,A -85,B 0,C 180,E1 -15132.655,E2 -15132.655} C_VEL
LIN {X 0,Y 337.423,Z 635.873,A -85,B 0,C 180,E1 -15133.325,E2 -15133.325} C_VEL
LIN {X 0,Y 337.832,Z 615.062,A -85,B 0,C 180,E1 -15134.018,E2 -15134.018} C_VEL
LIN {X 0,Y 338.67,Z 593.529,A -85,B 0,C 180,E1 -15134.642,E2 -15134.642} C_VEL
LIN {X 0,Y 333.155,Z 582.726,A -85,B 0,C 180,E1 -15135.825,E2 -15135.825} C_VEL
LIN {X 0,Y 327.584,Z 573.462,A -85,B 0,C 180,E1 -15137.081,E2 -15137.081} C_VEL
LIN {X 0,Y 324.819,Z 569.283,A -85,B 0,C 180,E1 -15137.749,E2 -15137.749} C_VEL
LIN {X 0,Y 322.809,Z 565.986,A -85,B 0,C 180,E1 -15138.266,E2 -15138.266} C_VEL
LIN {X 0,Y 320.362,Z 562.918,A -85,B 0,C 180,E1 -15138.877,E2 -15138.877} C_VEL
LIN {X 0,Y 319.665,Z 560.669,A -85,B 0,C 180,E1 -15139.16,E2 -15139.16} C_VEL
LIN {X 0,Y 319.567,Z 560.676,A -85,B 0,C 180,E1 -15143.32,E2 -15143.32} C_VEL
LIN {X 0,Y 319.632,Z 560.666,A -85,B 0,C 180,E1 -15146.089,E2 -15146.089} C_VEL
LIN {X 0,Y 319.588,Z 560.672,A -85,B 0,C 180,E1 -15148.934,E2 -15148.934} C_VEL
LIN {X 0,Y 319.53,Z 560.672,A -85,B 0,C 180,E1 -15151.863,E2 -15151.863} C_VEL
LIN {X 0,Y 319.578,Z 560.671,A -85,B 0,C 180,E1 -15155.544,E2 -15155.544} C_VEL
LIN {X 0,Y 319.571,Z 560.675,A -85,B 0,C 180,E1 -15158.009,E2 -15158.009} C_VEL
LIN {X 0,Y 319.524,Z 560.679,A -85,B 0,C 180,E1 -15161.598,E2 -15161.598} C_VEL
LIN {X 0,Y 319.515,Z 560.687,A -85,B 0,C 180,E1 -15165.263,E2 -15165.263} C_VEL
LIN {X 0,Y 319.527,Z 560.672,A -85,B 0,C 180,E1 -15168.713,E2 -15168.713} C_VEL
LIN {X 0,Y 319.631,Z 560.835,A -85,B 0,C 180,E1 -15170.201,E2 -15170.201} C_VEL
LIN {X 0,Y 322.452,Z 574.712,A -85,B 0,C 180,E1 -15174.337,E2 -15174.337} C_VEL
LIN {X 0,Y 324.547,Z 584.81,A -85,B 0,C 180,E1 -15177.224,E2 -15177.224} C_VEL
LIN {X 0,Y 323.18,Z 595.368,A -85,B 0,C 180,E1 -15179.99,E2 -15179.99} C_VEL
LIN {X 0,Y 323.901,Z 600.215,A -85,B 0,C 180,E1 -15180.34,E2 -15180.34} C_VEL
LIN {X 0,Y 324.619,Z 603.271,A -85,B 0,C 180,E1 -15180.604,E2 -15180.604} C_VEL
LIN {X 0,Y 327.83,Z 620.877,A -85,B 0,C 180,E1 -15181.897,E2 -15181.897} C_VEL
LIN {X 0,Y 330.795,Z 640.863,A -85,B 0,C 180,E1 -15183.168,E2 -15183.168} C_VEL
LIN {X 0,Y 331.663,Z 650.048,A -85,B 0,C 180,E1 -15183.656,E2 -15183.656} C_VEL
LIN {X 0,Y 334.167,Z 684.318,A -85,B 0,C 180,E1 -15185.289,E2 -15185.289} C_VEL
LIN {X 0,Y 332.26,Z 720.212,A -85,B 0,C 180,E1 -15186.429,E2 -15186.429} C_VEL
LIN {X 0,Y 330.847,Z 735.039,A -85,B 0,C 180,E1 -15187.108,E2 -15187.108} C_VEL
LIN {X 0,Y 328.962,Z 749.567,A -85,B 0,C 180,E1 -15188.046,E2 -15188.046} C_VEL
LIN {X 0,Y 327.152,Z 761.788,A -85,B 0,C 180,E1 -15189.076,E2 -15189.076} C_VEL
LIN {X 0,Y 325.047,Z 774.37,A -85,B 0,C 180,E1 -15190.42,E2 -15190.42} C_VEL
LIN {X 0,Y 323.122,Z 785.86,A -85,B 0,C 180,E1 -15191.945,E2 -15191.945} C_VEL
LIN {X 0,Y 321.627,Z 795.388,A -85,B 0,C 180,E1 -15193.498,E2 -15193.498} C_VEL
LIN {X 0,Y 320.323,Z 804.878,A -85,B 0,C 180,E1 -15195.399,E2 -15195.399} C_VEL
LIN {X 0,Y 319.372,Z 812.618,A -85,B 0,C 180,E1 -15197.288,E2 -15197.288} C_VEL
LIN {X 0,Y 318.798,Z 818.998,A -85,B 0,C 180,E1 -15199.201,E2 -15199.201} C_VEL
LIN {X 0,Y 318.68,Z 824.145,A -85,B 0,C 180,E1 -15201.12,E2 -15201.12} C_VEL
LIN {X 0,Y 318.722,Z 827.866,A -85,B 0,C 180,E1 -15202.878,E2 -15202.878} C_VEL
LIN {X 0,Y 319.111,Z 831.13,A -85,B 0,C 180,E1 -15204.947,E2 -15204.947} C_VEL
LIN {X 0,Y 319.344,Z 834.079,A -85,B 0,C 180,E1 -15207.478,E2 -15207.478} C_VEL
LIN {X 0,Y 319.461,Z 835.124,A -85,B 0,C 180,E1 -15208.74,E2 -15208.74} C_VEL
LIN {X 0,Y 319.641,Z 835.711,A -85,B 0,C 180,E1 -15210.001,E2 -15210.001} C_VEL
LIN {X 0,Y 319.341,Z 835.716,A -85,B 0,C 180,E1 -15211.262,E2 -15211.262} C_VEL
LIN {X 0,Y 319.12,Z 835.278,A -85,B 0,C 180,E1 -15212.525,E2 -15212.525} C_VEL
LIN {X 0,Y 319.033,Z 834.406,A -85,B 0,C 180,E1 -15213.79,E2 -15213.79} C_VEL
LIN {X 0,Y 318.86,Z 833.08,A -85,B 0,C 180,E1 -15215.059,E2 -15215.059} C_VEL
LIN {X 0,Y 318.618,Z 830.193,A -85,B 0,C 180,E1 -15216.971,E2 -15216.971} C_VEL
LIN {X 0,Y 318.522,Z 826.277,A -85,B 0,C 180,E1 -15218.886,E2 -15218.886} C_VEL
LIN {X 0,Y 318.678,Z 821.257,A -85,B 0,C 180,E1 -15220.805,E2 -15220.805} C_VEL
LIN {X 0,Y 319.421,Z 813.924,A -85,B 0,C 180,E1 -15223.034,E2 -15223.034} C_VEL
LIN {X 0,Y 320.398,Z 805.182,A -85,B 0,C 180,E1 -15225.169,E2 -15225.169} C_VEL
LIN {X 0,Y 322.112,Z 795.169,A -85,B 0,C 180,E1 -15227.131,E2 -15227.131} C_VEL
LIN {X 0,Y 324.386,Z 783.627,A -85,B 0,C 180,E1 -15228.965,E2 -15228.965} C_VEL
LIN {X 0,Y 326.553,Z 772.076,A -85,B 0,C 180,E1 -15230.471,E2 -15230.471} C_VEL
LIN {X 0,Y 328.838,Z 759.571,A -85,B 0,C 180,E1 -15231.799,E2 -15231.799} C_VEL
LIN {X 0,Y 331.232,Z 746.113,A -85,B 0,C 180,E1 -15232.948,E2 -15232.948} C_VEL
LIN {X 0,Y 333.718,Z 730.236,A -85,B 0,C 180,E1 -15233.999,E2 -15233.999} C_VEL
LIN {X 0,Y 335.719,Z 714.017,A -85,B 0,C 180,E1 -15234.804,E2 -15234.804} C_VEL
LIN {X 0,Y 337.538,Z 689.7,A -85,B 0,C 180,E1 -15235.665,E2 -15235.665} C_VEL
LIN {X 0,Y 337.837,Z 682.202,A -85,B 0,C 180,E1 -15235.944,E2 -15235.944} C_VEL
LIN {X 0,Y 337.75,Z 653.823,A -85,B 0,C 180,E1 -15237.223,E2 -15237.223} C_VEL
LIN {X 0,Y 336.644,Z 634.932,A -85,B 0,C 180,E1 -15238.3,E2 -15238.3} C_VEL
LIN {X 0,Y 334.831,Z 618.541,A -85,B 0,C 180,E1 -15239.456,E2 -15239.456} C_VEL
LIN {X 0,Y 332.542,Z 603.073,A -85,B 0,C 180,E1 -15240.755,E2 -15240.755} C_VEL
LIN {X 0,Y 330.418,Z 590.991,A -85,B 0,C 180,E1 -15241.943,E2 -15241.943} C_VEL
LIN {X 0,Y 329.278,Z 584.83,A -85,B 0,C 180,E1 -15242.607,E2 -15242.607} C_VEL
LIN {X 0,Y 327.881,Z 578.637,A -85,B 0,C 180,E1 -15243.376,E2 -15243.376} C_VEL
LIN {X 0,Y 324.518,Z 569.609,A -85,B 0,C 180,E1 -15245.026,E2 -15245.026} C_VEL
LIN {X 0,Y 323.591,Z 566.548,A -85,B 0,C 180,E1 -15245.587,E2 -15245.587} C_VEL
LIN {X 0,Y 322.769,Z 565.71,A -85,B 0,C 180,E1 -15245.953,E2 -15245.953} C_VEL
LIN {X 0,Y 320.656,Z 563.627,A -85,B 0,C 180,E1 -15246.929,E2 -15246.929} C_VEL
LIN {X 0,Y 319.626,Z 561.051,A -85,B 0,C 180,E1 -15247.632,E2 -15247.632} C_VEL
LIN {X 0,Y 319.57,Z 560.676,A -85,B 0,C 180,E1 -15247.777,E2 -15247.777} C_VEL
LIN {X 0,Y 319.53,Z 560.681,A -85,B 0,C 180,E1 -15251.597,E2 -15251.597} C_VEL
LIN {X 0,Y 319.493,Z 560.69,A -85,B 0,C 180,E1 -15255.257,E2 -15255.257} C_VEL
LIN {X 0,Y 319.533,Z 560.68,A -85,B 0,C 180,E1 -15258.712,E2 -15258.712} C_VEL
LIN {X 0,Y 319.566,Z 560.675,A -85,B 0,C 180,E1 -15262.348,E2 -15262.348} C_VEL
LIN {X 0,Y 319.586,Z 560.733,A -85,B 0,C 180,E1 -15264.073,E2 -15264.073} C_VEL
LIN {X 0,Y 320.246,Z 562.894,A -85,B 0,C 180,E1 -15264.566,E2 -15264.566} C_VEL
LIN {X 0,Y 322.132,Z 565.315,A -85,B 0,C 180,E1 -15265.486,E2 -15265.486} C_VEL
LIN {X 0,Y 323.847,Z 566.584,A -85,B 0,C 180,E1 -15266.178,E2 -15266.178} C_VEL
LIN {X 0,Y 325.537,Z 569.662,A -85,B 0,C 180,E1 -15266.922,E2 -15266.922} C_VEL
LIN {X 0,Y 327.673,Z 571.891,A -85,B 0,C 180,E1 -15267.69,E2 -15267.69} C_VEL
LIN {X 0,Y 330.086,Z 575.438,A -85,B 0,C 180,E1 -15268.527,E2 -15268.527} C_VEL
LIN {X 0,Y 331.295,Z 577.094,A -85,B 0,C 180,E1 -15268.92,E2 -15268.92} C_VEL
LIN {X 0,Y 334.619,Z 582.104,A -85,B 0,C 180,E1 -15269.929,E2 -15269.929} C_VEL
LIN {X 0,Y 338.865,Z 588.911,A -85,B 0,C 180,E1 -15271.098,E2 -15271.098} C_VEL
LIN {X 0,Y 343.57,Z 598.024,A -85,B 0,C 180,E1 -15272.319,E2 -15272.319} C_VEL
LIN {X 0,Y 342.868,Z 625.456,A -85,B 0,C 180,E1 -15273.239,E2 -15273.239} C_VEL
LIN {X 0,Y 342.325,Z 639.832,A -85,B 0,C 180,E1 -15273.939,E2 -15273.939} C_VEL
LIN {X 0,Y 341.266,Z 654.09,A -85,B 0,C 180,E1 -15274.865,E2 -15274.865} C_VEL
LIN {X 0,Y 339.864,Z 666.881,A -85,B 0,C 180,E1 -15275.92,E2 -15275.92} C_VEL
LIN {X 0,Y 338.168,Z 679.433,A -85,B 0,C 180,E1 -15277.227,E2 -15277.227} C_VEL
LIN {X 0,Y 335.985,Z 692.176,A -85,B 0,C 180,E1 -15278.848,E2 -15278.848} C_VEL
LIN {X 0,Y 334.114,Z 701.702,A -85,B 0,C 180,E1 -15280.332,E2 -15280.332} C_VEL
LIN {X 0,Y 331.972,Z 711.278,A -85,B 0,C 180,E1 -15282.123,E2 -15282.123} C_VEL
LIN {X 0,Y 329.631,Z 720.672,A -85,B 0,C 180,E1 -15284.268,E2 -15284.268} C_VEL
LIN {X 0,Y 327.645,Z 728.014,A -85,B 0,C 180,E1 -15286.352,E2 -15286.352} C_VEL
LIN {X 0,Y 325.614,Z 734.797,A -85,B 0,C 180,E1 -15288.798,E2 -15288.798} C_VEL
LIN {X 0,Y 323.818,Z 740.021,A -85,B 0,C 180,E1 -15291.261,E2 -15291.261} C_VEL
LIN {X 0,Y 322.626,Z 743.754,A -85,B 0,C 180,E1 -15293.746,E2 -15293.746} C_VEL
LIN {X 0,Y 321.512,Z 746.197,A -85,B 0,C 180,E1 -15296.239,E2 -15296.239} C_VEL
LIN {X 0,Y 320.796,Z 747.347,A -85,B 0,C 180,E1 -15298.744,E2 -15298.744} C_VEL
LIN {X 0,Y 320.31,Z 747.263,A -85,B 0,C 180,E1 -15301.257,E2 -15301.257} C_VEL
LIN {X 0,Y 319.975,Z 745.941,A -85,B 0,C 180,E1 -15303.778,E2 -15303.778} C_VEL
LIN {X 0,Y 319.801,Z 744.815,A -85,B 0,C 180,E1 -15305.042,E2 -15305.042} C_VEL
LIN {X 0,Y 320.093,Z 741.531,A -85,B 0,C 180,E1 -15307.569,E2 -15307.569} C_VEL
LIN {X 0,Y 320.283,Z 736.907,A -85,B 0,C 180,E1 -15310.11,E2 -15310.11} C_VEL
LIN {X 0,Y 320.718,Z 730.782,A -85,B 0,C 180,E1 -15312.658,E2 -15312.658} C_VEL
LIN {X 0,Y 321.391,Z 724.033,A -85,B 0,C 180,E1 -15314.888,E2 -15314.888} C_VEL
LIN {X 0,Y 322.206,Z 715.779,A -85,B 0,C 180,E1 -15317.125,E2 -15317.125} C_VEL
LIN {X 0,Y 323.234,Z 705.736,A -85,B 0,C 180,E1 -15319.364,E2 -15319.364} C_VEL
LIN {X 0,Y 324.387,Z 695.168,A -85,B 0,C 180,E1 -15321.311,E2 -15321.311} C_VEL
LIN {X 0,Y 325.475,Z 683.96,A -85,B 0,C 180,E1 -15323.039,E2 -15323.039} C_VEL
LIN {X 0,Y 326.719,Z 671.542,A -85,B 0,C 180,E1 -15324.63,E2 -15324.63} C_VEL
LIN {X 0,Y 327.751,Z 658.352,A -85,B 0,C 180,E1 -15326.03,E2 -15326.03} C_VEL
LIN {X 0,Y 328.762,Z 643.68,A -85,B 0,C 180,E1 -15327.275,E2 -15327.275} C_VEL
LIN {X 0,Y 329.566,Z 629.522,A -85,B 0,C 180,E1 -15328.214,E2 -15328.214} C_VEL
LIN {X 0,Y 330.153,Z 614.022,A -85,B 0,C 180,E1 -15328.982,E2 -15328.982} C_VEL
LIN {X 0,Y 330.424,Z 595.585,A -85,B 0,C 180,E1 -15329.6,E2 -15329.6} C_VEL
LIN {X 0,Y 330.344,Z 589.887,A -85,B 0,C 180,E1 -15329.777,E2 -15329.777} C_VEL
LIN {X 0,Y 319.563,Z 560.676,A -85,B 0,C 180,E1 -15331.306,E2 -15331.306} C_VEL
LIN {X 0,Y 319.561,Z 560.676,A -85,B 0,C 180,E1 -15334.876,E2 -15334.876} C_VEL
LIN {X 0,Y 319.574,Z 560.678,A -85,B 0,C 180,E1 -15338.007,E2 -15338.007} C_VEL
LIN {X 0,Y 319.526,Z 560.681,A -85,B 0,C 180,E1 -15341.596,E2 -15341.596} C_VEL
LIN {X 0,Y 319.488,Z 560.685,A -85,B 0,C 180,E1 -15345.256,E2 -15345.256} C_VEL
LIN {X 0,Y 319.528,Z 560.682,A -85,B 0,C 180,E1 -15348.711,E2 -15348.711} C_VEL
LIN {X 0,Y 319.578,Z 560.678,A -85,B 0,C 180,E1 -15352.343,E2 -15352.343} C_VEL
LIN {X 0,Y 319.56,Z 560.677,A -85,B 0,C 180,E1 -15355.123,E2 -15355.123} C_VEL
LIN {X 0,Y 319.565,Z 560.677,A -85,B 0,C 180,E1 -15359.058,E2 -15359.058} C_VEL
LIN {X 0,Y 319.605,Z 560.675,A -85,B 0,C 180,E1 -15362.497,E2 -15362.497} C_VEL
LIN {X 0,Y 319.604,Z 560.671,A -85,B 0,C 180,E1 -15365.303,E2 -15365.303} C_VEL
LIN {X 0,Y 319.596,Z 560.672,A -85,B 0,C 180,E1 -15368.047,E2 -15368.047} C_VEL
LIN {X 0,Y 319.688,Z 560.664,A -85,B 0,C 180,E1 -15370.961,E2 -15370.961} C_VEL
LIN {X 0,Y 319.729,Z 560.657,A -85,B 0,C 180,E1 -15375.275,E2 -15375.275} C_VEL
LIN {X 0,Y 319.756,Z 560.651,A -85,B 0,C 180,E1 -15379.872,E2 -15379.872} C_VEL
LIN {X 0,Y 319.931,Z 560.63,A -85,B 0,C 180,E1 -15382.425,E2 -15382.425} C_VEL
LIN {X 0,Y 319.747,Z 560.657,A -85,B 0,C 180,E1 -15384.955,E2 -15384.955} C_VEL
LIN {X 0,Y 319.99,Z 560.625,A -85,B 0,C 180,E1 -15387.482,E2 -15387.482} C_VEL
LIN {X 0,Y 320.148,Z 560.602,A -85,B 0,C 180,E1 -15389.999,E2 -15389.999} C_VEL
LIN {X 0,Y 319.99,Z 560.623,A -85,B 0,C 180,E1 -15392.517,E2 -15392.517} C_VEL
LIN {X 0,Y 319.948,Z 560.627,A -85,B 0,C 180,E1 -15396.305,E2 -15396.305} C_VEL
LIN {X 0,Y 319.84,Z 560.643,A -85,B 0,C 180,E1 -15398.847,E2 -15398.847} C_VEL
LIN {X 0,Y 319.682,Z 560.661,A -85,B 0,C 180,E1 -15402.699,E2 -15402.699} C_VEL
LIN {X 0,Y 319.696,Z 560.663,A -85,B 0,C 180,E1 -15405.295,E2 -15405.295} C_VEL
LIN {X 0,Y 319.67,Z 560.665,A -85,B 0,C 180,E1 -15409.254,E2 -15409.254} C_VEL
LIN {X 0,Y 319.566,Z 560.678,A -85,B 0,C 180,E1 -15413.319,E2 -15413.319} C_VEL
LIN {X 0,Y 319.631,Z 560.669,A -85,B 0,C 180,E1 -15416.087,E2 -15416.087} C_VEL
LIN {X 0,Y 319.586,Z 560.673,A -85,B 0,C 180,E1 -15418.933,E2 -15418.933} C_VEL
LIN {X 0,Y 319.534,Z 560.684,A -85,B 0,C 180,E1 -15421.86,E2 -15421.86} C_VEL
LIN {X 0,Y 319.576,Z 560.677,A -85,B 0,C 180,E1 -15425.543,E2 -15425.543} C_VEL
LIN {X 0,Y 319.593,Z 560.676,A -85,B 0,C 180,E1 -15428.004,E2 -15428.004} C_VEL
LIN {X 0,Y 319.567,Z 560.678,A -85,B 0,C 180,E1 -15431.606,E2 -15431.606} C_VEL
LIN {X 0,Y 319.627,Z 560.668,A -85,B 0,C 180,E1 -15435.283,E2 -15435.283} C_VEL
LIN {X 0,Y 319.578,Z 560.674,A -85,B 0,C 180,E1 -15438.72,E2 -15438.72} C_VEL
LIN {X 0,Y 319.617,Z 560.669,A -85,B 0,C 180,E1 -15441.313,E2 -15441.313} C_VEL
LIN {X 0,Y 329.368,Z 587.124,A -85,B 0,C 180,E1 -15442.638,E2 -15442.638} C_VEL
LIN {X 0,Y 328.584,Z 622.302,A -85,B 0,C 180,E1 -15443.617,E2 -15443.617} C_VEL
LIN {X 0,Y 328.308,Z 637.279,A -85,B 0,C 180,E1 -15444.274,E2 -15444.274} C_VEL
LIN {X 0,Y 327.595,Z 651.671,A -85,B 0,C 180,E1 -15445.167,E2 -15445.167} C_VEL
LIN {X 0,Y 327.158,Z 658.945,A -85,B 0,C 180,E1 -15445.733,E2 -15445.733} C_VEL
LIN {X 0,Y 326.25,Z 664.265,A -85,B 0,C 180,E1 -15446.164,E2 -15446.164} C_VEL
LIN {X 0,Y 322.95,Z 672.726,A -85,B 0,C 180,E1 -15446.852,E2 -15446.852} C_VEL
LIN {X 0,Y 319.411,Z 680.894,A -85,B 0,C 180,E1 -15447.64,E2 -15447.64} C_VEL
LIN {X 0,Y 318.153,Z 685.687,A -85,B 0,C 180,E1 -15448.224,E2 -15448.224} C_VEL
LIN {X 0,Y 317.112,Z 696.469,A -85,B 0,C 180,E1 -15449.805,E2 -15449.805} C_VEL
LIN {X 0,Y 316.142,Z 705.814,A -85,B 0,C 180,E1 -15451.449,E2 -15451.449} C_VEL
LIN {X 0,Y 315.148,Z 715.507,A -85,B 0,C 180,E1 -15453.513,E2 -15453.513} C_VEL
LIN {X 0,Y 314.304,Z 723.402,A -85,B 0,C 180,E1 -15455.565,E2 -15455.565} C_VEL
LIN {X 0,Y 313.652,Z 729.821,A -85,B 0,C 180,E1 -15457.61,E2 -15457.61} C_VEL
LIN {X 0,Y 313.196,Z 734.98,A -85,B 0,C 180,E1 -15459.647,E2 -15459.647} C_VEL
LIN {X 0,Y 312.858,Z 739.029,A -85,B 0,C 180,E1 -15461.67,E2 -15461.67} C_VEL
LIN {X 0,Y 312.703,Z 741.192,A -85,B 0,C 180,E1 -15463.012,E2 -15463.012} C_VEL
LIN {X 0,Y 312.686,Z 743.712,A -85,B 0,C 180,E1 -15465.119,E2 -15465.119} C_VEL
LIN {X 0,Y 312.781,Z 745.165,A -85,B 0,C 180,E1 -15467.016,E2 -15467.016} C_VEL
LIN {X 0,Y 313.14,Z 745.932,A -85,B 0,C 180,E1 -15469.657,E2 -15469.657} C_VEL
LIN {X 0,Y 313.417,Z 745.769,A -85,B 0,C 180,E1 -15470.97,E2 -15470.97} C_VEL
LIN {X 0,Y 313.715,Z 745.231,A -85,B 0,C 180,E1 -15472.276,E2 -15472.276} C_VEL
LIN {X 0,Y 314.713,Z 742.973,A -85,B 0,C 180,E1 -15474.876,E2 -15474.876} C_VEL
LIN {X 0,Y 315.898,Z 739.247,A -85,B 0,C 180,E1 -15477.45,E2 -15477.45} C_VEL
LIN {X 0,Y 317.045,Z 735.373,A -85,B 0,C 180,E1 -15479.366,E2 -15479.366} C_VEL
LIN {X 0,Y 318.374,Z 730.506,A -85,B 0,C 180,E1 -15481.265,E2 -15481.265} C_VEL
LIN {X 0,Y 320.082,Z 723.428,A -85,B 0,C 180,E1 -15483.462,E2 -15483.462} C_VEL
LIN {X 0,Y 321.942,Z 715.824,A -85,B 0,C 180,E1 -15485.324,E2 -15485.324} C_VEL
LIN {X 0,Y 323.842,Z 706.71,A -85,B 0,C 180,E1 -15487.169,E2 -15487.169} C_VEL
LIN {X 0,Y 325.72,Z 696.474,A -85,B 0,C 180,E1 -15488.844,E2 -15488.844} C_VEL
LIN {X 0,Y 327.583,Z 685.031,A -85,B 0,C 180,E1 -15490.352,E2 -15490.352} C_VEL
LIN {X 0,Y 329.123,Z 673.724,A -85,B 0,C 180,E1 -15491.549,E2 -15491.549} C_VEL
LIN {X 0,Y 330.415,Z 660.527,A -85,B 0,C 180,E1 -15492.671,E2 -15492.671} C_VEL
LIN {X 0,Y 331.314,Z 647.434,A -85,B 0,C 180,E1 -15493.52,E2 -15493.52} C_VEL
LIN {X 0,Y 331.848,Z 632.864,A -85,B 0,C 180,E1 -15494.198,E2 -15494.198} C_VEL
LIN {X 0,Y 332.859,Z 600.899,A -85,B 0,C 180,E1 -15495.19,E2 -15495.19} C_VEL
LIN {X 0,Y 333.007,Z 595.94,A -85,B 0,C 180,E1 -15495.348,E2 -15495.348} C_VEL
LIN {X 0,Y 327.661,Z 585.474,A -85,B 0,C 180,E1 -15496.582,E2 -15496.582} C_VEL
LIN {X 0,Y 322.446,Z 576.979,A -85,B 0,C 180,E1 -15497.844,E2 -15497.844} C_VEL
LIN {X 0,Y 318.344,Z 570.662,A -85,B 0,C 180,E1 -15498.917,E2 -15498.917} C_VEL
LIN {X 0,Y 316.162,Z 567.349,A -85,B 0,C 180,E1 -15499.533,E2 -15499.533} C_VEL
LIN {X 0,Y 315.478,Z 566.413,A -85,B 0,C 180,E1 -15499.727,E2 -15499.727} C_VEL
LIN {X 0,Y 313.428,Z 564.129,A -85,B 0,C 180,E1 -15500.293,E2 -15500.293} C_VEL
LIN {X 0,Y 312.57,Z 561.552,A -85,B 0,C 180,E1 -15500.659,E2 -15500.659} C_VEL
LIN {X 0,Y 312.54,Z 561.551,A -85,B 0,C 180,E1 -15503.877,E2 -15503.877} C_VEL
LIN {X 0,Y 312.581,Z 561.547,A -85,B 0,C 180,E1 -15506.724,E2 -15506.724} C_VEL
LIN {X 0,Y 312.543,Z 561.543,A -85,B 0,C 180,E1 -15509.651,E2 -15509.651} C_VEL
LIN {X 0,Y 312.517,Z 561.549,A -85,B 0,C 180,E1 -15513.69,E2 -15513.69} C_VEL
LIN {X 0,Y 312.524,Z 561.547,A -85,B 0,C 180,E1 -15517.386,E2 -15517.386} C_VEL
LIN {X 0,Y 312.488,Z 561.559,A -85,B 0,C 180,E1 -15520.71,E2 -15520.71} C_VEL
LIN {X 0,Y 312.471,Z 561.56,A -85,B 0,C 180,E1 -15524.207,E2 -15524.207} C_VEL
LIN {X 0,Y 312.485,Z 561.555,A -85,B 0,C 180,E1 -15527.919,E2 -15527.919} C_VEL
LIN {X 0,Y 312.574,Z 561.602,A -85,B 0,C 180,E1 -15529.974,E2 -15529.974} C_VEL
LIN {X 0,Y 314.835,Z 573.067,A -85,B 0,C 180,E1 -15533.478,E2 -15533.478} C_VEL
LIN {X 0,Y 317.311,Z 584.645,A -85,B 0,C 180,E1 -15536.887,E2 -15536.887} C_VEL
LIN {X 0,Y 317.259,Z 587.094,A -85,B 0,C 180,E1 -15537.572,E2 -15537.572} C_VEL
LIN {X 0,Y 316.734,Z 590.694,A -85,B 0,C 180,E1 -15538.549,E2 -15538.549} C_VEL
LIN {X 0,Y 317.409,Z 595.62,A -85,B 0,C 180,E1 -15538.934,E2 -15538.934} C_VEL
LIN {X 0,Y 318.257,Z 599.099,A -85,B 0,C 180,E1 -15539.274,E2 -15539.274} C_VEL
LIN {X 0,Y 320.953,Z 613.887,A -85,B 0,C 180,E1 -15540.471,E2 -15540.471} C_VEL
LIN {X 0,Y 323.336,Z 628.512,A -85,B 0,C 180,E1 -15541.532,E2 -15541.532} C_VEL
LIN {X 0,Y 325.846,Z 647.821,A -85,B 0,C 180,E1 -15542.759,E2 -15542.759} C_VEL
LIN {X 0,Y 328.326,Z 685.659,A -85,B 0,C 180,E1 -15544.629,E2 -15544.629} C_VEL
LIN {X 0,Y 326.385,Z 719.131,A -85,B 0,C 180,E1 -15545.722,E2 -15545.722} C_VEL
LIN {X 0,Y 324.85,Z 733.7,A -85,B 0,C 180,E1 -15546.408,E2 -15546.408} C_VEL
LIN {X 0,Y 323.023,Z 747.069,A -85,B 0,C 180,E1 -15547.284,E2 -15547.284} C_VEL
LIN {X 0,Y 320.809,Z 761.036,A -85,B 0,C 180,E1 -15548.474,E2 -15548.474} C_VEL
LIN {X 0,Y 318.579,Z 773.495,A -85,B 0,C 180,E1 -15549.838,E2 -15549.838} C_VEL
LIN {X 0,Y 316.565,Z 784.856,A -85,B 0,C 180,E1 -15551.39,E2 -15551.39} C_VEL
LIN {X 0,Y 314.8,Z 795.123,A -85,B 0,C 180,E1 -15553.129,E2 -15553.129} C_VEL
LIN {X 0,Y 313.355,Z 804.791,A -85,B 0,C 180,E1 -15555.143,E2 -15555.143} C_VEL
LIN {X 0,Y 312.401,Z 812.059,A -85,B 0,C 180,E1 -15557,E2 -15557} C_VEL
LIN {X 0,Y 311.756,Z 818.317,A -85,B 0,C 180,E1 -15558.954,E2 -15558.954} C_VEL
LIN {X 0,Y 311.596,Z 823.377,A -85,B 0,C 180,E1 -15560.917,E2 -15560.917} C_VEL
LIN {X 0,Y 311.641,Z 827.296,A -85,B 0,C 180,E1 -15562.876,E2 -15562.876} C_VEL
LIN {X 0,Y 312.032,Z 830.179,A -85,B 0,C 180,E1 -15564.832,E2 -15564.832} C_VEL
LIN {X 0,Y 312.35,Z 832.796,A -85,B 0,C 180,E1 -15567.422,E2 -15567.422} C_VEL
LIN {X 0,Y 312.471,Z 833.888,A -85,B 0,C 180,E1 -15568.712,E2 -15568.712} C_VEL
LIN {X 0,Y 312.632,Z 834.523,A -85,B 0,C 180,E1 -15570.001,E2 -15570.001} C_VEL
LIN {X 0,Y 312.328,Z 834.618,A -85,B 0,C 180,E1 -15571.29,E2 -15571.29} C_VEL
LIN {X 0,Y 312.08,Z 834.226,A -85,B 0,C 180,E1 -15572.582,E2 -15572.582} C_VEL
LIN {X 0,Y 311.983,Z 833.402,A -85,B 0,C 180,E1 -15573.876,E2 -15573.876} C_VEL
LIN {X 0,Y 311.786,Z 832.112,A -85,B 0,C 180,E1 -15575.174,E2 -15575.174} C_VEL
LIN {X 0,Y 311.54,Z 829.595,A -85,B 0,C 180,E1 -15576.974,E2 -15576.974} C_VEL
LIN {X 0,Y 311.437,Z 825.524,A -85,B 0,C 180,E1 -15579.09,E2 -15579.09} C_VEL
LIN {X 0,Y 311.648,Z 820.649,A -85,B 0,C 180,E1 -15581.052,E2 -15581.052} C_VEL
LIN {X 0,Y 312.434,Z 813.47,A -85,B 0,C 180,E1 -15583.331,E2 -15583.331} C_VEL
LIN {X 0,Y 313.615,Z 804.535,A -85,B 0,C 180,E1 -15585.6,E2 -15585.6} C_VEL
LIN {X 0,Y 315.325,Z 795.235,A -85,B 0,C 180,E1 -15587.512,E2 -15587.512} C_VEL
LIN {X 0,Y 317.708,Z 783.995,A -85,B 0,C 180,E1 -15589.38,E2 -15589.38} C_VEL
LIN {X 0,Y 320.189,Z 771.645,A -85,B 0,C 180,E1 -15591.066,E2 -15591.066} C_VEL
LIN {X 0,Y 322.62,Z 759.489,A -85,B 0,C 180,E1 -15592.41,E2 -15592.41} C_VEL
LIN {X 0,Y 325.468,Z 744.583,A -85,B 0,C 180,E1 -15593.715,E2 -15593.715} C_VEL
LIN {X 0,Y 327.887,Z 730.212,A -85,B 0,C 180,E1 -15594.707,E2 -15594.707} C_VEL
LIN {X 0,Y 330.13,Z 713.615,A -85,B 0,C 180,E1 -15595.569,E2 -15595.569} C_VEL
LIN {X 0,Y 331.741,Z 695.82,A -85,B 0,C 180,E1 -15596.245,E2 -15596.245} C_VEL
LIN {X 0,Y 332.456,Z 683.828,A -85,B 0,C 180,E1 -15596.678,E2 -15596.678} C_VEL
LIN {X 0,Y 332.577,Z 655.438,A -85,B 0,C 180,E1 -15598.005,E2 -15598.005} C_VEL
LIN {X 0,Y 331.726,Z 637.412,A -85,B 0,C 180,E1 -15599.065,E2 -15599.065} C_VEL
LIN {X 0,Y 330.089,Z 620.823,A -85,B 0,C 180,E1 -15600.279,E2 -15600.279} C_VEL
LIN {X 0,Y 327.971,Z 604.862,A -85,B 0,C 180,E1 -15601.678,E2 -15601.678} C_VEL
LIN {X 0,Y 326.123,Z 593.557,A -85,B 0,C 180,E1 -15602.855,E2 -15602.855} C_VEL
LIN {X 0,Y 325.309,Z 588.588,A -85,B 0,C 180,E1 -15603.409,E2 -15603.409} C_VEL
LIN {X 0,Y 324.161,Z 583.095,A -85,B 0,C 180,E1 -15604.13,E2 -15604.13} C_VEL
LIN {X 0,Y 321.138,Z 573.938,A -85,B 0,C 180,E1 -15605.836,E2 -15605.836} C_VEL
LIN {X 0,Y 320.672,Z 572.409,A -85,B 0,C 180,E1 -15606.138,E2 -15606.138} C_VEL
LIN {X 0,Y 318.406,Z 570.131,A -85,B 0,C 180,E1 -15607.24,E2 -15607.24} C_VEL
LIN {X 0,Y 317.073,Z 567.335,A -85,B 0,C 180,E1 -15608.138,E2 -15608.138} C_VEL
LIN {X 0,Y 314.274,Z 565.422,A -85,B 0,C 180,E1 -15609.905,E2 -15609.905} C_VEL
LIN {X 0,Y 312.745,Z 562.763,A -85,B 0,C 180,E1 -15611.469,E2 -15611.469} C_VEL
LIN {X 0,Y 312.491,Z 561.556,A -85,B 0,C 180,E1 -15612.004,E2 -15612.004} C_VEL
LIN {X 0,Y 312.463,Z 561.56,A -85,B 0,C 180,E1 -15616.035,E2 -15616.035} C_VEL
LIN {X 0,Y 312.518,Z 561.617,A -85,B 0,C 180,E1 -15619.933,E2 -15619.933} C_VEL
LIN {X 0,Y 313.461,Z 564.344,A -85,B 0,C 180,E1 -15621.167,E2 -15621.167} C_VEL
LIN {X 0,Y 315.783,Z 566.682,A -85,B 0,C 180,E1 -15622.865,E2 -15622.865} C_VEL
LIN {X 0,Y 317.253,Z 567.5,A -85,B 0,C 180,E1 -15623.664,E2 -15623.664} C_VEL
LIN {X 0,Y 318.807,Z 570.644,A -85,B 0,C 180,E1 -15624.653,E2 -15624.653} C_VEL
LIN {X 0,Y 321.316,Z 573.04,A -85,B 0,C 180,E1 -15625.78,E2 -15625.78} C_VEL
LIN {X 0,Y 323.3,Z 576.315,A -85,B 0,C 180,E1 -15626.676,E2 -15626.676} C_VEL
LIN {X 0,Y 324.866,Z 578.056,A -85,B 0,C 180,E1 -15627.259,E2 -15627.259} C_VEL
LIN {X 0,Y 327.433,Z 581.73,A -85,B 0,C 180,E1 -15628.198,E2 -15628.198} C_VEL
LIN {X 0,Y 331.284,Z 587.786,A -85,B 0,C 180,E1 -15629.467,E2 -15629.467} C_VEL
LIN {X 0,Y 335.595,Z 595.042,A -85,B 0,C 180,E1 -15630.738,E2 -15630.738} C_VEL
LIN {X 0,Y 338.583,Z 601.085,A -85,B 0,C 180,E1 -15631.549,E2 -15631.549} C_VEL
LIN {X 0,Y 337.69,Z 626.527,A -85,B 0,C 180,E1 -15632.441,E2 -15632.441} C_VEL
LIN {X 0,Y 337.132,Z 641.253,A -85,B 0,C 180,E1 -15633.162,E2 -15633.162} C_VEL
LIN {X 0,Y 335.994,Z 655.249,A -85,B 0,C 180,E1 -15634.085,E2 -15634.085} C_VEL
LIN {X 0,Y 334.475,Z 667.938,A -85,B 0,C 180,E1 -15635.15,E2 -15635.15} C_VEL
LIN {X 0,Y 332.624,Z 680.773,A -85,B 0,C 180,E1 -15636.496,E2 -15636.496} C_VEL
LIN {X 0,Y 330.512,Z 692.414,A -85,B 0,C 180,E1 -15637.989,E2 -15637.989} C_VEL
LIN {X 0,Y 328.291,Z 702.928,A -85,B 0,C 180,E1 -15639.642,E2 -15639.642} C_VEL
LIN {X 0,Y 325.996,Z 712.689,A -85,B 0,C 180,E1 -15641.49,E2 -15641.49} C_VEL
LIN {X 0,Y 323.575,Z 721.768,A -85,B 0,C 180,E1 -15643.598,E2 -15643.598} C_VEL
LIN {X 0,Y 321.644,Z 728.228,A -85,B 0,C 180,E1 -15645.446,E2 -15645.446} C_VEL
LIN {X 0,Y 319.443,Z 735.298,A -85,B 0,C 180,E1 -15647.935,E2 -15647.935} C_VEL
LIN {X 0,Y 317.462,Z 740.728,A -85,B 0,C 180,E1 -15650.442,E2 -15650.442} C_VEL
LIN {X 0,Y 316.431,Z 743.719,A -85,B 0,C 180,E1 -15652.341,E2 -15652.341} C_VEL
LIN {X 0,Y 315.154,Z 746.633,A -85,B 0,C 180,E1 -15654.882,E2 -15654.882} C_VEL
LIN {X 0,Y 314.19,Z 748.269,A -85,B 0,C 180,E1 -15657.435,E2 -15657.435} C_VEL
LIN {X 0,Y 313.549,Z 748.636,A -85,B 0,C 180,E1 -15659.999,E2 -15659.999} C_VEL
LIN {X 0,Y 313.038,Z 747.766,A -85,B 0,C 180,E1 -15662.573,E2 -15662.573} C_VEL
LIN {X 0,Y 312.771,Z 745.64,A -85,B 0,C 180,E1 -15665.156,E2 -15665.156} C_VEL
LIN {X 0,Y 312.986,Z 743.563,A -85,B 0,C 180,E1 -15666.792,E2 -15666.792} C_VEL
LIN {X 0,Y 313.123,Z 739.952,A -85,B 0,C 180,E1 -15669.039,E2 -15669.039} C_VEL
LIN {X 0,Y 313.467,Z 734.392,A -85,B 0,C 180,E1 -15671.641,E2 -15671.641} C_VEL
LIN {X 0,Y 314.074,Z 727.222,A -85,B 0,C 180,E1 -15674.249,E2 -15674.249} C_VEL
LIN {X 0,Y 314.814,Z 719.837,A -85,B 0,C 180,E1 -15676.412,E2 -15676.412} C_VEL
LIN {X 0,Y 315.91,Z 709.863,A -85,B 0,C 180,E1 -15678.818,E2 -15678.818} C_VEL
LIN {X 0,Y 316.991,Z 700.034,A -85,B 0,C 180,E1 -15680.777,E2 -15680.777} C_VEL
LIN {X 0,Y 318.222,Z 688.204,A -85,B 0,C 180,E1 -15682.736,E2 -15682.736} C_VEL
LIN {X 0,Y 319.348,Z 676.368,A -85,B 0,C 180,E1 -15684.37,E2 -15684.37} C_VEL
LIN {X 0,Y 320.479,Z 663.556,A -85,B 0,C 180,E1 -15685.837,E2 -15685.837} C_VEL
LIN {X 0,Y 321.565,Z 649.521,A -85,B 0,C 180,E1 -15687.144,E2 -15687.144} C_VEL
LIN {X 0,Y 322.44,Z 635.096,A -85,B 0,C 180,E1 -15688.209,E2 -15688.209} C_VEL
LIN {X 0,Y 323.199,Z 619.661,A -85,B 0,C 180,E1 -15689.072,E2 -15689.072} C_VEL
LIN {X 0,Y 323.467,Z 604.262,A -85,B 0,C 180,E1 -15689.685,E2 -15689.685} C_VEL
LIN {X 0,Y 323.494,Z 591.394,A -85,B 0,C 180,E1 -15690.09,E2 -15690.09} C_VEL
LIN {X 0,Y 312.509,Z 561.557,A -85,B 0,C 180,E1 -15691.665,E2 -15691.665} C_VEL
LIN {X 0,Y 312.507,Z 561.559,A -85,B 0,C 180,E1 -15694.209,E2 -15694.209} C_VEL
LIN {X 0,Y 312.535,Z 561.556,A -85,B 0,C 180,E1 -15698.089,E2 -15698.089} C_VEL
LIN {X 0,Y 312.484,Z 561.561,A -85,B 0,C 180,E1 -15702.08,E2 -15702.08} C_VEL
LIN {X 0,Y 312.458,Z 561.563,A -85,B 0,C 180,E1 -15706.034,E2 -15706.034} C_VEL
LIN {X 0,Y 312.49,Z 561.556,A -85,B 0,C 180,E1 -15709.29,E2 -15709.29} C_VEL
LIN {X 0,Y 312.538,Z 561.555,A -85,B 0,C 180,E1 -15712.616,E2 -15712.616} C_VEL
LIN {X 0,Y 312.519,Z 561.557,A -85,B 0,C 180,E1 -15716.31,E2 -15716.31} C_VEL
LIN {X 0,Y 312.537,Z 561.554,A -85,B 0,C 180,E1 -15720.348,E2 -15720.348} C_VEL
LIN {X 0,Y 312.596,Z 561.544,A -85,B 0,C 180,E1 -15724.066,E2 -15724.066} C_VEL
LIN {X 0,Y 312.586,Z 561.544,A -85,B 0,C 180,E1 -15727.528,E2 -15727.528} C_VEL
LIN {X 0,Y 312.637,Z 561.538,A -85,B 0,C 180,E1 -15731.656,E2 -15731.656} C_VEL
LIN {X 0,Y 312.692,Z 561.531,A -85,B 0,C 180,E1 -15735.685,E2 -15735.685} C_VEL
LIN {X 0,Y 312.7,Z 561.531,A -85,B 0,C 180,E1 -15739.641,E2 -15739.641} C_VEL
LIN {X 0,Y 312.87,Z 561.509,A -85,B 0,C 180,E1 -15742.253,E2 -15742.253} C_VEL
LIN {X 0,Y 312.717,Z 561.532,A -85,B 0,C 180,E1 -15744.842,E2 -15744.842} C_VEL
LIN {X 0,Y 312.989,Z 561.496,A -85,B 0,C 180,E1 -15748.713,E2 -15748.713} C_VEL
LIN {X 0,Y 312.989,Z 561.499,A -85,B 0,C 180,E1 -15751.286,E2 -15751.286} C_VEL
LIN {X 0,Y 312.716,Z 561.533,A -85,B 0,C 180,E1 -15755.157,E2 -15755.157} C_VEL
LIN {X 0,Y 312.868,Z 561.511,A -85,B 0,C 180,E1 -15757.745,E2 -15757.745} C_VEL
LIN {X 0,Y 312.669,Z 561.537,A -85,B 0,C 180,E1 -15761.67,E2 -15761.67} C_VEL
LIN {X 0,Y 312.696,Z 561.532,A -85,B 0,C 180,E1 -15764.887,E2 -15764.887} C_VEL
LIN {X 0,Y 312.626,Z 561.543,A -85,B 0,C 180,E1 -15769.236,E2 -15769.236} C_VEL
LIN {X 0,Y 312.542,Z 561.55,A -85,B 0,C 180,E1 -15772.789,E2 -15772.789} C_VEL
LIN {X 0,Y 312.599,Z 561.546,A -85,B 0,C 180,E1 -15775.935,E2 -15775.935} C_VEL
LIN {X 0,Y 312.542,Z 561.555,A -85,B 0,C 180,E1 -15779.649,E2 -15779.649} C_VEL
LIN {X 0,Y 312.515,Z 561.559,A -85,B 0,C 180,E1 -15783.689,E2 -15783.689} C_VEL
LIN {X 0,Y 312.548,Z 561.551,A -85,B 0,C 180,E1 -15787.381,E2 -15787.381} C_VEL
LIN {X 0,Y 312.497,Z 561.556,A -85,B 0,C 180,E1 -15790.707,E2 -15790.707} C_VEL
LIN {X 0,Y 312.573,Z 561.55,A -85,B 0,C 180,E1 -15794.187,E2 -15794.187} C_VEL
LIN {X 0,Y 312.55,Z 561.554,A -85,B 0,C 180,E1 -15797.904,E2 -15797.904} C_VEL
LIN {X 0,Y 312.571,Z 561.549,A -85,B 0,C 180,E1 -15800.933,E2 -15800.933} C_VEL
LIN {X 0,Y 318.258,Z 577.155,A -85,B 0,C 180,E1 -15801.746,E2 -15801.746} C_VEL
LIN {X 0,Y 322.521,Z 588.644,A -85,B 0,C 180,E1 -15802.316,E2 -15802.316} C_VEL
LIN {X 0,Y 321.782,Z 624.247,A -85,B 0,C 180,E1 -15803.349,E2 -15803.349} C_VEL
LIN {X 0,Y 321.409,Z 638.642,A -85,B 0,C 180,E1 -15804.002,E2 -15804.002} C_VEL
LIN {X 0,Y 320.719,Z 652.551,A -85,B 0,C 180,E1 -15804.885,E2 -15804.885} C_VEL
LIN {X 0,Y 319.862,Z 665.097,A -85,B 0,C 180,E1 -15805.925,E2 -15805.925} C_VEL
LIN {X 0,Y 318.853,Z 678.362,A -85,B 0,C 180,E1 -15807.316,E2 -15807.316} C_VEL
LIN {X 0,Y 318.153,Z 685.687,A -85,B 0,C 180,E1 -15808.224,E2 -15808.224} C_VEL
LIN {X 0,Y 316.921,Z 690.416,A -85,B 0,C 180,E1 -15808.838,E2 -15808.838} C_VEL
LIN {X 0,Y 313.377,Z 697.86,A -85,B 0,C 180,E1 -15809.853,E2 -15809.853} C_VEL
LIN {X 0,Y 309.955,Z 704.917,A -85,B 0,C 180,E1 -15810.957,E2 -15810.957} C_VEL
LIN {X 0,Y 308.883,Z 708.95,A -85,B 0,C 180,E1 -15811.72,E2 -15811.72} C_VEL
LIN {X 0,Y 308.039,Z 717.271,A -85,B 0,C 180,E1 -15813.584,E2 -15813.584} C_VEL
LIN {X 0,Y 307.206,Z 725.049,A -85,B 0,C 180,E1 -15815.683,E2 -15815.683} C_VEL
LIN {X 0,Y 306.541,Z 731.36,A -85,B 0,C 180,E1 -15817.773,E2 -15817.773} C_VEL
LIN {X 0,Y 306,Z 737.41,A -85,B 0,C 180,E1 -15820.329,E2 -15820.329} C_VEL
LIN {X 0,Y 305.701,Z 741.492,A -85,B 0,C 180,E1 -15822.611,E2 -15822.611} C_VEL
LIN {X 0,Y 305.671,Z 744.888,A -85,B 0,C 180,E1 -15825.351,E2 -15825.351} C_VEL
LIN {X 0,Y 305.729,Z 745.999,A -85,B 0,C 180,E1 -15826.711,E2 -15826.711} C_VEL
LIN {X 0,Y 306.093,Z 747.021,A -85,B 0,C 180,E1 -15829.416,E2 -15829.416} C_VEL
LIN {X 0,Y 306.668,Z 746.587,A -85,B 0,C 180,E1 -15832.097,E2 -15832.097} C_VEL
LIN {X 0,Y 307.699,Z 744.682,A -85,B 0,C 180,E1 -15834.759,E2 -15834.759} C_VEL
LIN {X 0,Y 308.925,Z 741.241,A -85,B 0,C 180,E1 -15837.393,E2 -15837.393} C_VEL
LIN {X 0,Y 310.555,Z 736.184,A -85,B 0,C 180,E1 -15840.001,E2 -15840.001} C_VEL
LIN {X 0,Y 311.997,Z 731.206,A -85,B 0,C 180,E1 -15841.937,E2 -15841.937} C_VEL
LIN {X 0,Y 313.571,Z 725.156,A -85,B 0,C 180,E1 -15843.856,E2 -15843.856} C_VEL
LIN {X 0,Y 315.538,Z 717.717,A -85,B 0,C 180,E1 -15845.753,E2 -15845.753} C_VEL
LIN {X 0,Y 317.558,Z 708.744,A -85,B 0,C 180,E1 -15847.631,E2 -15847.631} C_VEL
LIN {X 0,Y 319.526,Z 698.669,A -85,B 0,C 180,E1 -15849.336,E2 -15849.336} C_VEL
LIN {X 0,Y 321.716,Z 686.234,A -85,B 0,C 180,E1 -15851.02,E2 -15851.02} C_VEL
LIN {X 0,Y 323.351,Z 675.027,A -85,B 0,C 180,E1 -15852.235,E2 -15852.235} C_VEL
LIN {X 0,Y 324.722,Z 661.835,A -85,B 0,C 180,E1 -15853.375,E2 -15853.375} C_VEL
LIN {X 0,Y 325.689,Z 648.497,A -85,B 0,C 180,E1 -15854.249,E2 -15854.249} C_VEL
LIN {X 0,Y 326.249,Z 633.789,A -85,B 0,C 180,E1 -15854.942,E2 -15854.942} C_VEL
LIN {X 0,Y 327.54,Z 600.102,A -85,B 0,C 180,E1 -15856.026,E2 -15856.026} C_VEL
LIN {X 0,Y 327.458,Z 598.356,A -85,B 0,C 180,E1 -15856.108,E2 -15856.108} C_VEL
LIN {X 0,Y 322.887,Z 589.502,A -85,B 0,C 180,E1 -15857.223,E2 -15857.223} C_VEL
LIN {X 0,Y 317.281,Z 580.153,A -85,B 0,C 180,E1 -15858.679,E2 -15858.679} C_VEL
LIN {X 0,Y 314.048,Z 575.331,A -85,B 0,C 180,E1 -15859.585,E2 -15859.585} C_VEL
LIN {X 0,Y 311.915,Z 572.12,A -85,B 0,C 180,E1 -15860.217,E2 -15860.217} C_VEL
LIN {X 0,Y 309.702,Z 569.202,A -85,B 0,C 180,E1 -15860.897,E2 -15860.897} C_VEL
LIN {X 0,Y 308.981,Z 567.665,A -85,B 0,C 180,E1 -15861.163,E2 -15861.163} C_VEL
LIN {X 0,Y 306.747,Z 565.62,A -85,B 0,C 180,E1 -15861.847,E2 -15861.847} C_VEL
LIN {X 0,Y 305.629,Z 563.016,A -85,B 0,C 180,E1 -15862.298,E2 -15862.298} C_VEL
LIN {X 0,Y 305.554,Z 562.426,A -85,B 0,C 180,E1 -15862.393,E2 -15862.393} C_VEL
LIN {X 0,Y 305.551,Z 562.421,A -85,B 0,C 180,E1 -15866.23,E2 -15866.23} C_VEL
LIN {X 0,Y 305.494,Z 562.426,A -85,B 0,C 180,E1 -15869.051,E2 -15869.051} C_VEL
LIN {X 0,Y 305.463,Z 562.429,A -85,B 0,C 180,E1 -15873.518,E2 -15873.518} C_VEL
LIN {X 0,Y 305.473,Z 562.425,A -85,B 0,C 180,E1 -15876.74,E2 -15876.74} C_VEL
LIN {X 0,Y 305.453,Z 562.435,A -85,B 0,C 180,E1 -15880.601,E2 -15880.601} C_VEL
LIN {X 0,Y 305.417,Z 562.438,A -85,B 0,C 180,E1 -15884.494,E2 -15884.494} C_VEL
LIN {X 0,Y 305.445,Z 562.429,A -85,B 0,C 180,E1 -15888.145,E2 -15888.145} C_VEL
LIN {X 0,Y 305.51,Z 562.461,A -85,B 0,C 180,E1 -15889.776,E2 -15889.776} C_VEL
LIN {X 0,Y 307.94,Z 574.699,A -85,B 0,C 180,E1 -15893.603,E2 -15893.603} C_VEL
LIN {X 0,Y 310.322,Z 585.872,A -85,B 0,C 180,E1 -15896.926,E2 -15896.926} C_VEL
LIN {X 0,Y 311.419,Z 592.116,A -85,B 0,C 180,E1 -15897.525,E2 -15897.525} C_VEL
LIN {X 0,Y 312.085,Z 594.933,A -85,B 0,C 180,E1 -15897.827,E2 -15897.827} C_VEL
LIN {X 0,Y 313.2,Z 600.738,A -85,B 0,C 180,E1 -15898.366,E2 -15898.366} C_VEL
LIN {X 0,Y 315.785,Z 615.629,A -85,B 0,C 180,E1 -15899.637,E2 -15899.637} C_VEL
LIN {X 0,Y 318.626,Z 634.359,A -85,B 0,C 180,E1 -15901.034,E2 -15901.034} C_VEL
LIN {X 0,Y 320.506,Z 651.346,A -85,B 0,C 180,E1 -15902.104,E2 -15902.104} C_VEL
LIN {X 0,Y 322.547,Z 686.926,A -85,B 0,C 180,E1 -15903.921,E2 -15903.921} C_VEL
LIN {X 0,Y 320.638,Z 716.92,A -85,B 0,C 180,E1 -15904.925,E2 -15904.925} C_VEL
LIN {X 0,Y 318.922,Z 732.521,A -85,B 0,C 180,E1 -15905.682,E2 -15905.682} C_VEL
LIN {X 0,Y 316.872,Z 746.79,A -85,B 0,C 180,E1 -15906.644,E2 -15906.644} C_VEL
LIN {X 0,Y 314.87,Z 758.906,A -85,B 0,C 180,E1 -15907.702,E2 -15907.702} C_VEL
LIN {X 0,Y 312.414,Z 771.446,A -85,B 0,C 180,E1 -15909.077,E2 -15909.077} C_VEL
LIN {X 0,Y 310.033,Z 783.937,A -85,B 0,C 180,E1 -15910.811,E2 -15910.811} C_VEL
LIN {X 0,Y 308.261,Z 793.293,A -85,B 0,C 180,E1 -15912.418,E2 -15912.418} C_VEL
LIN {X 0,Y 306.466,Z 803.441,A -85,B 0,C 180,E1 -15914.567,E2 -15914.567} C_VEL
LIN {X 0,Y 305.414,Z 811.533,A -85,B 0,C 180,E1 -15916.697,E2 -15916.697} C_VEL
LIN {X 0,Y 304.729,Z 817.657,A -85,B 0,C 180,E1 -15918.696,E2 -15918.696} C_VEL
LIN {X 0,Y 304.507,Z 822.594,A -85,B 0,C 180,E1 -15920.703,E2 -15920.703} C_VEL
LIN {X 0,Y 304.579,Z 826.652,A -85,B 0,C 180,E1 -15922.844,E2 -15922.844} C_VEL
LIN {X 0,Y 304.935,Z 829.252,A -85,B 0,C 180,E1 -15924.711,E2 -15924.711} C_VEL
LIN {X 0,Y 305.35,Z 831.497,A -85,B 0,C 180,E1 -15927.362,E2 -15927.362} C_VEL
LIN {X 0,Y 305.477,Z 832.639,A -85,B 0,C 180,E1 -15928.682,E2 -15928.682} C_VEL
LIN {X 0,Y 305.626,Z 833.321,A -85,B 0,C 180,E1 -15930.001,E2 -15930.001} C_VEL
LIN {X 0,Y 305.311,Z 833.467,A -85,B 0,C 180,E1 -15931.32,E2 -15931.32} C_VEL
LIN {X 0,Y 305.042,Z 833.165,A -85,B 0,C 180,E1 -15932.642,E2 -15932.642} C_VEL
LIN {X 0,Y 304.931,Z 832.399,A -85,B 0,C 180,E1 -15933.966,E2 -15933.966} C_VEL
LIN {X 0,Y 304.693,Z 831.159,A -85,B 0,C 180,E1 -15935.295,E2 -15935.295} C_VEL
LIN {X 0,Y 304.476,Z 828.956,A -85,B 0,C 180,E1 -15936.999,E2 -15936.999} C_VEL
LIN {X 0,Y 304.34,Z 824.797,A -85,B 0,C 180,E1 -15939.303,E2 -15939.303} C_VEL
LIN {X 0,Y 304.608,Z 820.039,A -85,B 0,C 180,E1 -15941.311,E2 -15941.311} C_VEL
LIN {X 0,Y 305.436,Z 813.069,A -85,B 0,C 180,E1 -15943.642,E2 -15943.642} C_VEL
LIN {X 0,Y 306.76,Z 804.346,A -85,B 0,C 180,E1 -15945.958,E2 -15945.958} C_VEL
LIN {X 0,Y 308.57,Z 795.297,A -85,B 0,C 180,E1 -15947.908,E2 -15947.908} C_VEL
LIN {X 0,Y 311.041,Z 784.483,A -85,B 0,C 180,E1 -15949.812,E2 -15949.812} C_VEL
LIN {X 0,Y 313.635,Z 772.548,A -85,B 0,C 180,E1 -15951.527,E2 -15951.527} C_VEL
LIN {X 0,Y 316.461,Z 759.513,A -85,B 0,C 180,E1 -15953.043,E2 -15953.043} C_VEL
LIN {X 0,Y 319.416,Z 745.177,A -85,B 0,C 180,E1 -15954.366,E2 -15954.366} C_VEL
LIN {X 0,Y 322.316,Z 729.292,A -85,B 0,C 180,E1 -15955.509,E2 -15955.509} C_VEL
LIN {X 0,Y 324.711,Z 713.089,A -85,B 0,C 180,E1 -15956.384,E2 -15956.384} C_VEL
LIN {X 0,Y 326.438,Z 696.044,A -85,B 0,C 180,E1 -15957.073,E2 -15957.073} C_VEL
LIN {X 0,Y 327.177,Z 684.823,A -85,B 0,C 180,E1 -15957.493,E2 -15957.493} C_VEL
LIN {X 0,Y 327.548,Z 656.677,A -85,B 0,C 180,E1 -15958.851,E2 -15958.851} C_VEL
LIN {X 0,Y 326.907,Z 639.315,A -85,B 0,C 180,E1 -15959.911,E2 -15959.911} C_VEL
LIN {X 0,Y 325.476,Z 622.612,A -85,B 0,C 180,E1 -15961.182,E2 -15961.182} C_VEL
LIN {X 0,Y 323.546,Z 606.132,A -85,B 0,C 180,E1 -15962.699,E2 -15962.699} C_VEL
LIN {X 0,Y 321.543,Z 592.336,A -85,B 0,C 180,E1 -15964.239,E2 -15964.239} C_VEL
LIN {X 0,Y 320.637,Z 587.731,A -85,B 0,C 180,E1 -15964.874,E2 -15964.874} C_VEL
LIN {X 0,Y 317.866,Z 578.565,A -85,B 0,C 180,E1 -15966.654,E2 -15966.654} C_VEL
LIN {X 0,Y 315.751,Z 575.961,A -85,B 0,C 180,E1 -15967.831,E2 -15967.831} C_VEL
LIN {X 0,Y 314.679,Z 573.893,A -85,B 0,C 180,E1 -15968.584,E2 -15968.584} C_VEL
LIN {X 0,Y 312.046,Z 571.724,A -85,B 0,C 180,E1 -15970.459,E2 -15970.459} C_VEL
LIN {X 0,Y 310.82,Z 568.973,A -85,B 0,C 180,E1 -15971.989,E2 -15971.989} C_VEL
LIN {X 0,Y 310.601,Z 568.372,A -85,B 0,C 180,E1 -15972.358,E2 -15972.358} C_VEL
LIN {X 0,Y 309.181,Z 567.873,A -85,B 0,C 180,E1 -15975.197,E2 -15975.197} C_VEL
LIN {X 0,Y 309.567,Z 568.029,A -85,B 0,C 180,E1 -15977.852,E2 -15977.852} C_VEL
LIN {X 0,Y 310.794,Z 568.609,A -85,B 0,C 180,E1 -15979.682,E2 -15979.682} C_VEL
LIN {X 0,Y 311.97,Z 571.501,A -85,B 0,C 180,E1 -15981.177,E2 -15981.177} C_VEL
LIN {X 0,Y 314.306,Z 573.676,A -85,B 0,C 180,E1 -15982.862,E2 -15982.862} C_VEL
LIN {X 0,Y 315.08,Z 574.2,A -85,B 0,C 180,E1 -15983.322,E2 -15983.322} C_VEL
LIN {X 0,Y 317.017,Z 577.604,A -85,B 0,C 180,E1 -15984.512,E2 -15984.512} C_VEL
LIN {X 0,Y 318.893,Z 579.598,A -85,B 0,C 180,E1 -15985.41,E2 -15985.41} C_VEL
LIN {X 0,Y 321.161,Z 583.027,A -85,B 0,C 180,E1 -15986.459,E2 -15986.459} C_VEL
LIN {X 0,Y 322.557,Z 584.993,A -85,B 0,C 180,E1 -15987.014,E2 -15987.014} C_VEL
LIN {X 0,Y 325.333,Z 589.143,A -85,B 0,C 180,E1 -15988.064,E2 -15988.064} C_VEL
LIN {X 0,Y 328.915,Z 594.861,A -85,B 0,C 180,E1 -15989.28,E2 -15989.28} C_VEL
LIN {X 0,Y 333.065,Z 602.653,A -85,B 0,C 180,E1 -15990.555,E2 -15990.555} C_VEL
LIN {X 0,Y 333.649,Z 603.945,A -85,B 0,C 180,E1 -15990.739,E2 -15990.739} C_VEL
LIN {X 0,Y 332.695,Z 629.81,A -85,B 0,C 180,E1 -15991.683,E2 -15991.683} C_VEL
LIN {X 0,Y 331.924,Z 644.414,A -85,B 0,C 180,E1 -15992.448,E2 -15992.448} C_VEL
LIN {X 0,Y 330.747,Z 657.345,A -85,B 0,C 180,E1 -15993.344,E2 -15993.344} C_VEL
LIN {X 0,Y 328.977,Z 670.986,A -85,B 0,C 180,E1 -15994.519,E2 -15994.519} C_VEL
LIN {X 0,Y 326.984,Z 683.528,A -85,B 0,C 180,E1 -15995.897,E2 -15995.897} C_VEL
LIN {X 0,Y 324.51,Z 695.929,A -85,B 0,C 180,E1 -15997.56,E2 -15997.56} C_VEL
LIN {X 0,Y 322.197,Z 706.118,A -85,B 0,C 180,E1 -15999.239,E2 -15999.239} C_VEL
LIN {X 0,Y 319.809,Z 715.188,A -85,B 0,C 180,E1 -16001.046,E2 -16001.046} C_VEL
LIN {X 0,Y 317.169,Z 724.246,A -85,B 0,C 180,E1 -16003.258,E2 -16003.258} C_VEL
LIN {X 0,Y 315.135,Z 730.582,A -85,B 0,C 180,E1 -16005.139,E2 -16005.139} C_VEL
LIN {X 0,Y 313.332,Z 735.787,A -85,B 0,C 180,E1 -16007.038,E2 -16007.038} C_VEL
LIN {X 0,Y 311.2,Z 741.37,A -85,B 0,C 180,E1 -16009.591,E2 -16009.591} C_VEL
LIN {X 0,Y 310.272,Z 743.61,A -85,B 0,C 180,E1 -16010.876,E2 -16010.876} C_VEL
LIN {X 0,Y 308.886,Z 746.973,A -85,B 0,C 180,E1 -16013.467,E2 -16013.467} C_VEL
LIN {X 0,Y 307.646,Z 749.06,A -85,B 0,C 180,E1 -16016.07,E2 -16016.07} C_VEL
LIN {X 0,Y 306.852,Z 749.866,A -85,B 0,C 180,E1 -16018.687,E2 -16018.687} C_VEL
LIN {X 0,Y 306.278,Z 749.437,A -85,B 0,C 180,E1 -16021.314,E2 -16021.314} C_VEL
LIN {X 0,Y 305.93,Z 747.758,A -85,B 0,C 180,E1 -16023.951,E2 -16023.951} C_VEL
LIN {X 0,Y 305.741,Z 746.455,A -85,B 0,C 180,E1 -16025.275,E2 -16025.275} C_VEL
LIN {X 0,Y 305.967,Z 744.496,A -85,B 0,C 180,E1 -16026.789,E2 -16026.789} C_VEL
LIN {X 0,Y 306.093,Z 740.485,A -85,B 0,C 180,E1 -16029.248,E2 -16029.248} C_VEL
LIN {X 0,Y 306.466,Z 734.727,A -85,B 0,C 180,E1 -16031.91,E2 -16031.91} C_VEL
LIN {X 0,Y 306.997,Z 728.314,A -85,B 0,C 180,E1 -16034.246,E2 -16034.246} C_VEL
LIN {X 0,Y 307.862,Z 720.194,A -85,B 0,C 180,E1 -16036.653,E2 -16036.653} C_VEL
LIN {X 0,Y 308.892,Z 710.878,A -85,B 0,C 180,E1 -16038.918,E2 -16038.918} C_VEL
LIN {X 0,Y 309.985,Z 701.002,A -85,B 0,C 180,E1 -16040.921,E2 -16040.921} C_VEL
LIN {X 0,Y 311.228,Z 689.115,A -85,B 0,C 180,E1 -16042.925,E2 -16042.925} C_VEL
LIN {X 0,Y 312.411,Z 677.224,A -85,B 0,C 180,E1 -16044.593,E2 -16044.593} C_VEL
LIN {X 0,Y 313.507,Z 665.342,A -85,B 0,C 180,E1 -16045.987,E2 -16045.987} C_VEL
LIN {X 0,Y 314.559,Z 652.196,A -85,B 0,C 180,E1 -16047.259,E2 -16047.259} C_VEL
LIN {X 0,Y 315.451,Z 638.183,A -85,B 0,C 180,E1 -16048.347,E2 -16048.347} C_VEL
LIN {X 0,Y 316.203,Z 622.579,A -85,B 0,C 180,E1 -16049.273,E2 -16049.273} C_VEL
LIN {X 0,Y 316.623,Z 607.006,A -85,B 0,C 180,E1 -16049.929,E2 -16049.929} C_VEL
LIN {X 0,Y 316.652,Z 592.949,A -85,B 0,C 180,E1 -16050.388,E2 -16050.388} C_VEL
LIN {X 0,Y 305.462,Z 562.454,A -85,B 0,C 180,E1 -16052.055,E2 -16052.055} C_VEL
LIN {X 0,Y 305.463,Z 562.432,A -85,B 0,C 180,E1 -16055.112,E2 -16055.112} C_VEL
LIN {X 0,Y 305.467,Z 562.434,A -85,B 0,C 180,E1 -16058.532,E2 -16058.532} C_VEL
LIN {X 0,Y 305.455,Z 562.436,A -85,B 0,C 180,E1 -16062.585,E2 -16062.585} C_VEL
LIN {X 0,Y 305.473,Z 562.43,A -85,B 0,C 180,E1 -16067.41,E2 -16067.41} C_VEL
LIN {X 0,Y 305.495,Z 562.428,A -85,B 0,C 180,E1 -16071.6,E2 -16071.6} C_VEL
LIN {X 0,Y 305.463,Z 562.434,A -85,B 0,C 180,E1 -16074.886,E2 -16074.886} C_VEL
LIN {X 0,Y 305.449,Z 562.437,A -85,B 0,C 180,E1 -16078.355,E2 -16078.355} C_VEL
LIN {X 0,Y 305.512,Z 562.427,A -85,B 0,C 180,E1 -16081.112,E2 -16081.112} C_VEL
LIN {X 0,Y 305.564,Z 562.42,A -85,B 0,C 180,E1 -16084.087,E2 -16084.087} C_VEL
LIN {X 0,Y 305.5,Z 562.429,A -85,B 0,C 180,E1 -16088.402,E2 -16088.402} C_VEL
LIN {X 0,Y 305.589,Z 562.418,A -85,B 0,C 180,E1 -16091.217,E2 -16091.217} C_VEL
LIN {X 0,Y 305.647,Z 562.41,A -85,B 0,C 180,E1 -16095.348,E2 -16095.348} C_VEL
LIN {X 0,Y 305.637,Z 562.412,A -85,B 0,C 180,E1 -16099.399,E2 -16099.399} C_VEL
LIN {X 0,Y 305.811,Z 562.388,A -85,B 0,C 180,E1 -16102.074,E2 -16102.074} C_VEL
LIN {X 0,Y 305.688,Z 562.406,A -85,B 0,C 180,E1 -16104.723,E2 -16104.723} C_VEL
LIN {X 0,Y 305.955,Z 562.372,A -85,B 0,C 180,E1 -16108.683,E2 -16108.683} C_VEL
LIN {X 0,Y 305.955,Z 562.374,A -85,B 0,C 180,E1 -16111.315,E2 -16111.315} C_VEL
LIN {X 0,Y 305.849,Z 562.384,A -85,B 0,C 180,E1 -16116.597,E2 -16116.597} C_VEL
LIN {X 0,Y 305.733,Z 562.404,A -85,B 0,C 180,E1 -16119.259,E2 -16119.259} C_VEL
LIN {X 0,Y 305.588,Z 562.421,A -85,B 0,C 180,E1 -16123.295,E2 -16123.295} C_VEL
LIN {X 0,Y 305.59,Z 562.417,A -85,B 0,C 180,E1 -16126.019,E2 -16126.019} C_VEL
LIN {X 0,Y 305.573,Z 562.423,A -85,B 0,C 180,E1 -16129.444,E2 -16129.444} C_VEL
LIN {X 0,Y 305.487,Z 562.43,A -85,B 0,C 180,E1 -16133.041,E2 -16133.041} C_VEL
LIN {X 0,Y 305.543,Z 562.423,A -85,B 0,C 180,E1 -16136.227,E2 -16136.227} C_VEL
LIN {X 0,Y 305.492,Z 562.429,A -85,B 0,C 180,E1 -16139.05,E2 -16139.05} C_VEL
LIN {X 0,Y 305.444,Z 562.438,A -85,B 0,C 180,E1 -16141.951,E2 -16141.951} C_VEL
LIN {X 0,Y 305.458,Z 562.433,A -85,B 0,C 180,E1 -16145.113,E2 -16145.113} C_VEL
LIN {X 0,Y 305.487,Z 562.43,A -85,B 0,C 180,E1 -16148.539,E2 -16148.539} C_VEL
LIN {X 0,Y 305.498,Z 562.428,A -85,B 0,C 180,E1 -16152.596,E2 -16152.596} C_VEL
LIN {X 0,Y 305.525,Z 562.427,A -85,B 0,C 180,E1 -16156.364,E2 -16156.364} C_VEL
LIN {X 0,Y 305.527,Z 562.426,A -85,B 0,C 180,E1 -16160.507,E2 -16160.507} C_VEL
LIN {X 0,Y 315.712,Z 590.414,A -85,B 0,C 180,E1 -16161.994,E2 -16161.994} C_VEL
LIN {X 0,Y 314.968,Z 624.395,A -85,B 0,C 180,E1 -16163.001,E2 -16163.001} C_VEL
LIN {X 0,Y 314.553,Z 639.693,A -85,B 0,C 180,E1 -16163.702,E2 -16163.702} C_VEL
